LIN {X 0,Y 216.52,Z 296.519,A -85,B 0,C 180,E1 -21835.267,E2 -21835.267} C_VEL
LIN {X 0,Y 214.915,Z 310.205,A -85,B 0,C 180,E1 -21836.01,E2 -21836.01} C_VEL
LIN {X 0,Y 213.159,Z 322.237,A -85,B 0,C 180,E1 -21837.044,E2 -21837.044} C_VEL
LIN {X 0,Y 210.843,Z 333.547,A -85,B 0,C 180,E1 -21838.334,E2 -21838.334} C_VEL
LIN {X 0,Y 208.05,Z 345.191,A -85,B 0,C 180,E1 -21840.117,E2 -21840.117} C_VEL
LIN {X 0,Y 205.01,Z 355.654,A -85,B 0,C 180,E1 -21842.157,E2 -21842.157} C_VEL
LIN {X 0,Y 202.418,Z 364.207,A -85,B 0,C 180,E1 -21844.281,E2 -21844.281} C_VEL
LIN {X 0,Y 199.781,Z 372.178,A -85,B 0,C 180,E1 -21846.724,E2 -21846.724} C_VEL
LIN {X 0,Y 197.037,Z 379.781,A -85,B 0,C 180,E1 -21849.651,E2 -21849.651} C_VEL
LIN {X 0,Y 194.335,Z 386.855,A -85,B 0,C 180,E1 -21853.184,E2 -21853.184} C_VEL
LIN {X 0,Y 192.658,Z 391.564,A -85,B 0,C 180,E1 -21856.285,E2 -21856.285} C_VEL
LIN {X 0,Y 191.459,Z 395.168,A -85,B 0,C 180,E1 -21859.425,E2 -21859.425} C_VEL
LIN {X 0,Y 190.867,Z 397.03,A -85,B 0,C 180,E1 -21861.531,E2 -21861.531} C_VEL
LIN {X 0,Y 190.523,Z 398.428,A -85,B 0,C 180,E1 -21863.647,E2 -21863.647} C_VEL
LIN {X 0,Y 190.151,Z 400.035,A -85,B 0,C 180,E1 -21867.883,E2 -21867.883} C_VEL
LIN {X 0,Y 190.161,Z 400.264,A -85,B 0,C 180,E1 -21870.001,E2 -21870.001} C_VEL
LIN {X 0,Y 190.151,Z 400.068,A -85,B 0,C 180,E1 -21872.119,E2 -21872.119} C_VEL
LIN {X 0,Y 190.277,Z 399.478,A -85,B 0,C 180,E1 -21874.237,E2 -21874.237} C_VEL
LIN {X 0,Y 190.523,Z 398.504,A -85,B 0,C 180,E1 -21876.354,E2 -21876.354} C_VEL
LIN {X 0,Y 190.863,Z 397.139,A -85,B 0,C 180,E1 -21878.471,E2 -21878.471} C_VEL
LIN {X 0,Y 191.808,Z 394.255,A -85,B 0,C 180,E1 -21881.627,E2 -21881.627} C_VEL
LIN {X 0,Y 193.155,Z 390.346,A -85,B 0,C 180,E1 -21884.756,E2 -21884.756} C_VEL
LIN {X 0,Y 194.985,Z 385.304,A -85,B 0,C 180,E1 -21887.841,E2 -21887.841} C_VEL
LIN {X 0,Y 197.437,Z 378.955,A -85,B 0,C 180,E1 -21890.853,E2 -21890.853} C_VEL
LIN {X 0,Y 200.011,Z 371.649,A -85,B 0,C 180,E1 -21893.599,E2 -21893.599} C_VEL
LIN {X 0,Y 202.794,Z 362.923,A -85,B 0,C 180,E1 -21896.223,E2 -21896.223} C_VEL
LIN {X 0,Y 205.882,Z 353.047,A -85,B 0,C 180,E1 -21898.549,E2 -21898.549} C_VEL
LIN {X 0,Y 209.005,Z 341.929,A -85,B 0,C 180,E1 -21900.57,E2 -21900.57} C_VEL
LIN {X 0,Y 211.513,Z 331.031,A -85,B 0,C 180,E1 -21902.116,E2 -21902.116} C_VEL
LIN {X 0,Y 213.783,Z 318.986,A -85,B 0,C 180,E1 -21903.411,E2 -21903.411} C_VEL
LIN {X 0,Y 215.659,Z 305.842,A -85,B 0,C 180,E1 -21904.403,E2 -21904.403} C_VEL
LIN {X 0,Y 216.816,Z 292.984,A -85,B 0,C 180,E1 -21905.015,E2 -21905.015} C_VEL
LIN {X 0,Y 219.192,Z 241.525,A -85,B 0,C 180,E1 -21906.632,E2 -21906.632} C_VEL
LIN {X 0,Y 214.01,Z 228.643,A -85,B 0,C 180,E1 -21908.209,E2 -21908.209} C_VEL
LIN {X 0,Y 207.201,Z 214.231,A -85,B 0,C 180,E1 -21910.349,E2 -21910.349} C_VEL
LIN {X 0,Y 200.702,Z 202.668,A -85,B 0,C 180,E1 -21912.494,E2 -21912.494} C_VEL
LIN {X 0,Y 197.748,Z 198.045,A -85,B 0,C 180,E1 -21913.511,E2 -21913.511} C_VEL
LIN {X 0,Y 195.588,Z 194.613,A -85,B 0,C 180,E1 -21914.288,E2 -21914.288} C_VEL
LIN {X 0,Y 193.261,Z 191.834,A -85,B 0,C 180,E1 -21915.109,E2 -21915.109} C_VEL
LIN {X 0,Y 192.615,Z 190.071,A -85,B 0,C 180,E1 -21915.548,E2 -21915.548} C_VEL
LIN {X 0,Y 192.511,Z 189.538,A -85,B 0,C 180,E1 -21916.081,E2 -21916.081} C_VEL
LIN {X 0,Y 192.519,Z 189.499,A -85,B 0,C 180,E1 -21920.051,E2 -21920.051} C_VEL
LIN {X 0,Y 192.56,Z 189.439,A -85,B 0,C 180,E1 -21924.27,E2 -21924.27} C_VEL
LIN {X 0,Y 192.61,Z 189.447,A -85,B 0,C 180,E1 -21927.058,E2 -21927.058} C_VEL
LIN {X 0,Y 192.665,Z 189.47,A -85,B 0,C 180,E1 -21931.692,E2 -21931.692} C_VEL
LIN {X 0,Y 192.685,Z 189.474,A -85,B 0,C 180,E1 -21936.346,E2 -21936.346} C_VEL
LIN {X 0,Y 192.731,Z 189.477,A -85,B 0,C 180,E1 -21941.458,E2 -21941.458} C_VEL
LIN {X 0,Y 192.851,Z 189.461,A -85,B 0,C 180,E1 -21947.37,E2 -21947.37} C_VEL
LIN {X 0,Y 193.06,Z 189.411,A -85,B 0,C 180,E1 -21951.627,E2 -21951.627} C_VEL
LIN {X 0,Y 193.259,Z 189.386,A -85,B 0,C 180,E1 -21957.916,E2 -21957.916} C_VEL
LIN {X 0,Y 193.438,Z 189.382,A -85,B 0,C 180,E1 -21960,E2 -21960} C_VEL
LIN {X 0,Y 192.963,Z 189.423,A -85,B 0,C 180,E1 -21964.177,E2 -21964.177} C_VEL
LIN {X 0,Y 193.025,Z 189.441,A -85,B 0,C 180,E1 -21968.374,E2 -21968.374} C_VEL
LIN {X 0,Y 192.789,Z 189.451,A -85,B 0,C 180,E1 -21972.634,E2 -21972.634} C_VEL
LIN {X 0,Y 192.745,Z 189.456,A -85,B 0,C 180,E1 -21976.96,E2 -21976.96} C_VEL
LIN {X 0,Y 192.611,Z 189.492,A -85,B 0,C 180,E1 -21981.4,E2 -21981.4} C_VEL
LIN {X 0,Y 192.646,Z 189.469,A -85,B 0,C 180,E1 -21984.213,E2 -21984.213} C_VEL
LIN {X 0,Y 192.644,Z 189.473,A -85,B 0,C 180,E1 -21988.889,E2 -21988.889} C_VEL
LIN {X 0,Y 192.596,Z 189.478,A -85,B 0,C 180,E1 -21993.186,E2 -21993.186} C_VEL
LIN {X 0,Y 192.55,Z 189.454,A -85,B 0,C 180,E1 -21998.352,E2 -21998.352} C_VEL
LIN {X 0,Y 192.546,Z 189.606,A -85,B 0,C 180,E1 -22003.258,E2 -22003.258} C_VEL
LIN {X 0,Y 193.232,Z 191.826,A -85,B 0,C 180,E1 -22004.713,E2 -22004.713} C_VEL
LIN {X 0,Y 195.599,Z 195.89,A -85,B 0,C 180,E1 -22005.696,E2 -22005.696} C_VEL
LIN {X 0,Y 202.058,Z 206.618,A -85,B 0,C 180,E1 -22007.96,E2 -22007.96} C_VEL
LIN {X 0,Y 208.446,Z 218.785,A -85,B 0,C 180,E1 -22010.059,E2 -22010.059} C_VEL
LIN {X 0,Y 214.326,Z 231.789,A -85,B 0,C 180,E1 -22011.905,E2 -22011.905} C_VEL
LIN {X 0,Y 217.009,Z 238.438,A -85,B 0,C 180,E1 -22012.729,E2 -22012.729} C_VEL
LIN {X 0,Y 217.391,Z 241.526,A -85,B 0,C 180,E1 -22012.93,E2 -22012.93} C_VEL
LIN {X 0,Y 216.613,Z 246.06,A -85,B 0,C 180,E1 -22012.96,E2 -22012.96} C_VEL
LIN {X 0,Y 213.129,Z 256.558,A -85,B 0,C 180,E1 -22012.687,E2 -22012.687} C_VEL
LIN {X 0,Y 212.744,Z 259.307,A -85,B 0,C 180,E1 -22012.722,E2 -22012.722} C_VEL
LIN {X 0,Y 210.674,Z 300.138,A -85,B 0,C 180,E1 -22014.065,E2 -22014.065} C_VEL
LIN {X 0,Y 209.14,Z 313.363,A -85,B 0,C 180,E1 -22014.813,E2 -22014.813} C_VEL
LIN {X 0,Y 206.891,Z 326.323,A -85,B 0,C 180,E1 -22015.91,E2 -22015.91} C_VEL
LIN {X 0,Y 204.512,Z 337.393,A -85,B 0,C 180,E1 -22017.232,E2 -22017.232} C_VEL
LIN {X 0,Y 201.553,Z 348.935,A -85,B 0,C 180,E1 -22019.048,E2 -22019.048} C_VEL
LIN {X 0,Y 198.374,Z 359.328,A -85,B 0,C 180,E1 -22021.137,E2 -22021.137} C_VEL
LIN {X 0,Y 195.51,Z 367.823,A -85,B 0,C 180,E1 -22023.299,E2 -22023.299} C_VEL
LIN {X 0,Y 192.771,Z 375.975,A -85,B 0,C 180,E1 -22025.913,E2 -22025.913} C_VEL
LIN {X 0,Y 189.944,Z 383.312,A -85,B 0,C 180,E1 -22028.853,E2 -22028.853} C_VEL
LIN {X 0,Y 187.139,Z 390.37,A -85,B 0,C 180,E1 -22032.515,E2 -22032.515} C_VEL
LIN {X 0,Y 185.395,Z 395.063,A -85,B 0,C 180,E1 -22035.735,E2 -22035.735} C_VEL
LIN {X 0,Y 184.159,Z 398.646,A -85,B 0,C 180,E1 -22038.999,E2 -22038.999} C_VEL
LIN {X 0,Y 183.61,Z 400.493,A -85,B 0,C 180,E1 -22041.192,E2 -22041.192} C_VEL
LIN {X 0,Y 183.297,Z 401.878,A -85,B 0,C 180,E1 -22043.394,E2 -22043.394} C_VEL
LIN {X 0,Y 183.032,Z 403.227,A -85,B 0,C 180,E1 -22046.698,E2 -22046.698} C_VEL
LIN {X 0,Y 183.065,Z 403.678,A -85,B 0,C 180,E1 -22049.999,E2 -22049.999} C_VEL
LIN {X 0,Y 183.032,Z 403.215,A -85,B 0,C 180,E1 -22053.3,E2 -22053.3} C_VEL
LIN {X 0,Y 183.297,Z 401.849,A -85,B 0,C 180,E1 -22056.604,E2 -22056.604} C_VEL
LIN {X 0,Y 183.612,Z 400.45,A -85,B 0,C 180,E1 -22058.806,E2 -22058.806} C_VEL
LIN {X 0,Y 184.507,Z 397.518,A -85,B 0,C 180,E1 -22062.092,E2 -22062.092} C_VEL
LIN {X 0,Y 185.875,Z 393.55,A -85,B 0,C 180,E1 -22065.346,E2 -22065.346} C_VEL
LIN {X 0,Y 188.255,Z 387.448,A -85,B 0,C 180,E1 -22069.065,E2 -22069.065} C_VEL
LIN {X 0,Y 190.832,Z 380.783,A -85,B 0,C 180,E1 -22072.177,E2 -22072.177} C_VEL
LIN {X 0,Y 193.536,Z 373.421,A -85,B 0,C 180,E1 -22074.905,E2 -22074.905} C_VEL
LIN {X 0,Y 196.714,Z 364.027,A -85,B 0,C 180,E1 -22077.673,E2 -22077.673} C_VEL
LIN {X 0,Y 200.047,Z 353.54,A -85,B 0,C 180,E1 -22080.04,E2 -22080.04} C_VEL
LIN {X 0,Y 202.948,Z 343.16,A -85,B 0,C 180,E1 -22081.875,E2 -22081.875} C_VEL
LIN {X 0,Y 205.721,Z 331.768,A -85,B 0,C 180,E1 -22083.425,E2 -22083.425} C_VEL
LIN {X 0,Y 207.911,Z 320.025,A -85,B 0,C 180,E1 -22084.631,E2 -22084.631} C_VEL
LIN {X 0,Y 209.832,Z 306.994,A -85,B 0,C 180,E1 -22085.544,E2 -22085.544} C_VEL
LIN {X 0,Y 210.927,Z 294.034,A -85,B 0,C 180,E1 -22086.129,E2 -22086.129} C_VEL
LIN {X 0,Y 213.185,Z 246.397,A -85,B 0,C 180,E1 -22087.649,E2 -22087.649} C_VEL
LIN {X 0,Y 211.994,Z 242.409,A -85,B 0,C 180,E1 -22088.065,E2 -22088.065} C_VEL
LIN {X 0,Y 205.399,Z 226.595,A -85,B 0,C 180,E1 -22090.22,E2 -22090.22} C_VEL
LIN {X 0,Y 199.419,Z 214.433,A -85,B 0,C 180,E1 -22092.261,E2 -22092.261} C_VEL
LIN {X 0,Y 193.932,Z 204.867,A -85,B 0,C 180,E1 -22094.229,E2 -22094.229} C_VEL
LIN {X 0,Y 191.078,Z 200.191,A -85,B 0,C 180,E1 -22095.309,E2 -22095.309} C_VEL
LIN {X 0,Y 188.425,Z 196.048,A -85,B 0,C 180,E1 -22096.352,E2 -22096.352} C_VEL
LIN {X 0,Y 185.757,Z 191.777,A -85,B 0,C 180,E1 -22097.545,E2 -22097.545} C_VEL
LIN {X 0,Y 185.478,Z 190.463,A -85,B 0,C 180,E1 -22098.394,E2 -22098.394} C_VEL
LIN {X 0,Y 185.5,Z 190.321,A -85,B 0,C 180,E1 -22102.711,E2 -22102.711} C_VEL
LIN {X 0,Y 185.536,Z 190.375,A -85,B 0,C 180,E1 -22107.973,E2 -22107.973} C_VEL
LIN {X 0,Y 185.575,Z 190.352,A -85,B 0,C 180,E1 -22110.576,E2 -22110.576} C_VEL
LIN {X 0,Y 185.574,Z 190.35,A -85,B 0,C 180,E1 -22115.381,E2 -22115.381} C_VEL
LIN {X 0,Y 185.651,Z 190.339,A -85,B 0,C 180,E1 -22121.149,E2 -22121.149} C_VEL
LIN {X 0,Y 185.678,Z 190.354,A -85,B 0,C 180,E1 -22124.636,E2 -22124.636} C_VEL
LIN {X 0,Y 185.918,Z 190.303,A -85,B 0,C 180,E1 -22129.359,E2 -22129.359} C_VEL
LIN {X 0,Y 185.951,Z 190.307,A -85,B 0,C 180,E1 -22133.49,E2 -22133.49} C_VEL
LIN {X 0,Y 186.197,Z 190.285,A -85,B 0,C 180,E1 -22137.837,E2 -22137.837} C_VEL
LIN {X 0,Y 186.399,Z 190.259,A -85,B 0,C 180,E1 -22140,E2 -22140} C_VEL
LIN {X 0,Y 185.913,Z 190.313,A -85,B 0,C 180,E1 -22144.336,E2 -22144.336} C_VEL
LIN {X 0,Y 186.002,Z 190.289,A -85,B 0,C 180,E1 -22148.693,E2 -22148.693} C_VEL
LIN {X 0,Y 185.757,Z 190.344,A -85,B 0,C 180,E1 -22153.121,E2 -22153.121} C_VEL
LIN {X 0,Y 185.688,Z 190.356,A -85,B 0,C 180,E1 -22158.885,E2 -22158.885} C_VEL
LIN {X 0,Y 185.596,Z 190.366,A -85,B 0,C 180,E1 -22164.663,E2 -22164.663} C_VEL
LIN {X 0,Y 185.574,Z 190.361,A -85,B 0,C 180,E1 -22169.494,E2 -22169.494} C_VEL
LIN {X 0,Y 185.494,Z 190.318,A -85,B 0,C 180,E1 -22174.633,E2 -22174.633} C_VEL
LIN {X 0,Y 185.5,Z 190.331,A -85,B 0,C 180,E1 -22177.315,E2 -22177.315} C_VEL
LIN {X 0,Y 185.448,Z 190.501,A -85,B 0,C 180,E1 -22182.077,E2 -22182.077} C_VEL
LIN {X 0,Y 185.683,Z 191.483,A -85,B 0,C 180,E1 -22182.632,E2 -22182.632} C_VEL
LIN {X 0,Y 187.311,Z 194.335,A -85,B 0,C 180,E1 -22183.371,E2 -22183.371} C_VEL
LIN {X 0,Y 188.847,Z 195.941,A -85,B 0,C 180,E1 -22183.95,E2 -22183.95} C_VEL
LIN {X 0,Y 191.21,Z 199.43,A -85,B 0,C 180,E1 -22184.865,E2 -22184.865} C_VEL
LIN {X 0,Y 195.417,Z 205.792,A -85,B 0,C 180,E1 -22186.412,E2 -22186.412} C_VEL
LIN {X 0,Y 201.414,Z 216.342,A -85,B 0,C 180,E1 -22188.514,E2 -22188.514} C_VEL
LIN {X 0,Y 207.913,Z 229.985,A -85,B 0,C 180,E1 -22190.684,E2 -22190.684} C_VEL
LIN {X 0,Y 213.386,Z 243.368,A -85,B 0,C 180,E1 -22192.44,E2 -22192.44} C_VEL
LIN {X 0,Y 210.73,Z 296.676,A -85,B 0,C 180,E1 -22194.173,E2 -22194.173} C_VEL
LIN {X 0,Y 209.058,Z 310.386,A -85,B 0,C 180,E1 -22194.931,E2 -22194.931} C_VEL
LIN {X 0,Y 207.054,Z 323.393,A -85,B 0,C 180,E1 -22196.089,E2 -22196.089} C_VEL
LIN {X 0,Y 204.484,Z 335.201,A -85,B 0,C 180,E1 -22197.521,E2 -22197.521} C_VEL
LIN {X 0,Y 201.532,Z 346.551,A -85,B 0,C 180,E1 -22199.337,E2 -22199.337} C_VEL
LIN {X 0,Y 198.444,Z 356.78,A -85,B 0,C 180,E1 -22201.44,E2 -22201.44} C_VEL
LIN {X 0,Y 195.424,Z 366.126,A -85,B 0,C 180,E1 -22203.921,E2 -22203.921} C_VEL
LIN {X 0,Y 192.291,Z 374.888,A -85,B 0,C 180,E1 -22206.867,E2 -22206.867} C_VEL
LIN {X 0,Y 189.533,Z 382.075,A -85,B 0,C 180,E1 -22209.942,E2 -22209.942} C_VEL
LIN {X 0,Y 187.528,Z 386.921,A -85,B 0,C 180,E1 -22212.555,E2 -22212.555} C_VEL
LIN {X 0,Y 185.75,Z 391.631,A -85,B 0,C 180,E1 -22215.764,E2 -22215.764} C_VEL
LIN {X 0,Y 184.461,Z 395.234,A -85,B 0,C 180,E1 -22219.019,E2 -22219.019} C_VEL
LIN {X 0,Y 183.832,Z 397.096,A -85,B 0,C 180,E1 -22221.205,E2 -22221.205} C_VEL
LIN {X 0,Y 183.448,Z 398.494,A -85,B 0,C 180,E1 -22223.401,E2 -22223.401} C_VEL
LIN {X 0,Y 183.097,Z 399.767,A -85,B 0,C 180,E1 -22226.367,E2 -22226.367} C_VEL
LIN {X 0,Y 183.072,Z 400.329,A -85,B 0,C 180,E1 -22230.001,E2 -22230.001} C_VEL
LIN {X 0,Y 183.154,Z 399.723,A -85,B 0,C 180,E1 -22233.906,E2 -22233.906} C_VEL
LIN {X 0,Y 183.448,Z 398.569,A -85,B 0,C 180,E1 -22236.6,E2 -22236.6} C_VEL
LIN {X 0,Y 183.829,Z 397.204,A -85,B 0,C 180,E1 -22238.797,E2 -22238.797} C_VEL
LIN {X 0,Y 184.841,Z 394.319,A -85,B 0,C 180,E1 -22242.071,E2 -22242.071} C_VEL
LIN {X 0,Y 186.272,Z 390.41,A -85,B 0,C 180,E1 -22245.315,E2 -22245.315} C_VEL
LIN {X 0,Y 188.219,Z 385.368,A -85,B 0,C 180,E1 -22248.505,E2 -22248.505} C_VEL
LIN {X 0,Y 190.8,Z 379.018,A -85,B 0,C 180,E1 -22251.614,E2 -22251.614} C_VEL
LIN {X 0,Y 193.325,Z 372.255,A -85,B 0,C 180,E1 -22254.258,E2 -22254.258} C_VEL
LIN {X 0,Y 196.444,Z 362.985,A -85,B 0,C 180,E1 -22257.139,E2 -22257.139} C_VEL
LIN {X 0,Y 199.684,Z 353.109,A -85,B 0,C 180,E1 -22259.521,E2 -22259.521} C_VEL
LIN {X 0,Y 202.918,Z 341.989,A -85,B 0,C 180,E1 -22261.591,E2 -22261.591} C_VEL
LIN {X 0,Y 205.529,Z 331.09,A -85,B 0,C 180,E1 -22263.169,E2 -22263.169} C_VEL
LIN {X 0,Y 207.889,Z 319.043,A -85,B 0,C 180,E1 -22264.49,E2 -22264.49} C_VEL
LIN {X 0,Y 209.796,Z 306.311,A -85,B 0,C 180,E1 -22265.474,E2 -22265.474} C_VEL
LIN {X 0,Y 211.048,Z 293.249,A -85,B 0,C 180,E1 -22266.109,E2 -22266.109} C_VEL
LIN {X 0,Y 213.46,Z 243.344,A -85,B 0,C 180,E1 -22267.711,E2 -22267.711} C_VEL
LIN {X 0,Y 208.208,Z 230.53,A -85,B 0,C 180,E1 -22269.397,E2 -22269.397} C_VEL
LIN {X 0,Y 202.113,Z 217.696,A -85,B 0,C 180,E1 -22271.426,E2 -22271.426} C_VEL
LIN {X 0,Y 196.616,Z 207.676,A -85,B 0,C 180,E1 -22273.349,E2 -22273.349} C_VEL
LIN {X 0,Y 193.586,Z 202.92,A -85,B 0,C 180,E1 -22274.445,E2 -22274.445} C_VEL
LIN {X 0,Y 191.026,Z 199.227,A -85,B 0,C 180,E1 -22275.397,E2 -22275.397} C_VEL
LIN {X 0,Y 188.755,Z 195.702,A -85,B 0,C 180,E1 -22276.292,E2 -22276.292} C_VEL
LIN {X 0,Y 186.317,Z 192.945,A -85,B 0,C 180,E1 -22277.236,E2 -22277.236} C_VEL
LIN {X 0,Y 185.532,Z 190.905,A -85,B 0,C 180,E1 -22277.792,E2 -22277.792} C_VEL
LIN {X 0,Y 185.452,Z 190.446,A -85,B 0,C 180,E1 -22278.233,E2 -22278.233} C_VEL
LIN {X 0,Y 185.506,Z 190.333,A -85,B 0,C 180,E1 -22282.712,E2 -22282.712} C_VEL
LIN {X 0,Y 185.546,Z 190.342,A -85,B 0,C 180,E1 -22287.975,E2 -22287.975} C_VEL
LIN {X 0,Y 185.582,Z 190.361,A -85,B 0,C 180,E1 -22290.576,E2 -22290.576} C_VEL
LIN {X 0,Y 185.58,Z 190.369,A -85,B 0,C 180,E1 -22295.381,E2 -22295.381} C_VEL
LIN {X 0,Y 185.674,Z 190.357,A -85,B 0,C 180,E1 -22301.134,E2 -22301.134} C_VEL
LIN {X 0,Y 185.762,Z 190.342,A -85,B 0,C 180,E1 -22306.879,E2 -22306.879} C_VEL
LIN {X 0,Y 186.008,Z 190.288,A -85,B 0,C 180,E1 -22311.307,E2 -22311.307} C_VEL
LIN {X 0,Y 186.204,Z 190.264,A -85,B 0,C 180,E1 -22317.837,E2 -22317.837} C_VEL
LIN {X 0,Y 186.402,Z 190.258,A -85,B 0,C 180,E1 -22320,E2 -22320} C_VEL
LIN {X 0,Y 185.909,Z 190.301,A -85,B 0,C 180,E1 -22324.336,E2 -22324.336} C_VEL
LIN {X 0,Y 185.974,Z 190.317,A -85,B 0,C 180,E1 -22328.694,E2 -22328.694} C_VEL
LIN {X 0,Y 185.717,Z 190.337,A -85,B 0,C 180,E1 -22333.124,E2 -22333.124} C_VEL
LIN {X 0,Y 185.683,Z 190.333,A -85,B 0,C 180,E1 -22337.626,E2 -22337.626} C_VEL
LIN {X 0,Y 185.574,Z 190.358,A -85,B 0,C 180,E1 -22342.254,E2 -22342.254} C_VEL
LIN {X 0,Y 185.558,Z 190.372,A -85,B 0,C 180,E1 -22347.033,E2 -22347.033} C_VEL
LIN {X 0,Y 185.577,Z 190.352,A -85,B 0,C 180,E1 -22349.493,E2 -22349.493} C_VEL
LIN {X 0,Y 185.498,Z 190.333,A -85,B 0,C 180,E1 -22354.632,E2 -22354.632} C_VEL
LIN {X 0,Y 185.504,Z 190.321,A -85,B 0,C 180,E1 -22357.314,E2 -22357.314} C_VEL
LIN {X 0,Y 185.476,Z 190.553,A -85,B 0,C 180,E1 -22361.606,E2 -22361.606} C_VEL
LIN {X 0,Y 185.867,Z 192.023,A -85,B 0,C 180,E1 -22362.424,E2 -22362.424} C_VEL
LIN {X 0,Y 189.734,Z 197.961,A -85,B 0,C 180,E1 -22364.054,E2 -22364.054} C_VEL
LIN {X 0,Y 195.512,Z 207.366,A -85,B 0,C 180,E1 -22366.245,E2 -22366.245} C_VEL
LIN {X 0,Y 202.294,Z 219.885,A -85,B 0,C 180,E1 -22368.637,E2 -22368.637} C_VEL
LIN {X 0,Y 208.335,Z 233.114,A -85,B 0,C 180,E1 -22370.661,E2 -22370.661} C_VEL
LIN {X 0,Y 213.143,Z 245.402,A -85,B 0,C 180,E1 -22372.226,E2 -22372.226} C_VEL
LIN {X 0,Y 213.37,Z 248.029,A -85,B 0,C 180,E1 -22372.382,E2 -22372.382} C_VEL
LIN {X 0,Y 212.744,Z 259.307,A -85,B 0,C 180,E1 -22372.722,E2 -22372.722} C_VEL
LIN {X 0,Y 211.928,Z 265.149,A -85,B 0,C 180,E1 -22372.798,E2 -22372.798} C_VEL
LIN {X 0,Y 206.47,Z 284.171,A -85,B 0,C 180,E1 -22372.463,E2 -22372.463} C_VEL
LIN {X 0,Y 205.612,Z 290.015,A -85,B 0,C 180,E1 -22372.531,E2 -22372.531} C_VEL
LIN {X 0,Y 204.494,Z 304.483,A -85,B 0,C 180,E1 -22373.099,E2 -22373.099} C_VEL
LIN {X 0,Y 202.62,Z 318.008,A -85,B 0,C 180,E1 -22374.021,E2 -22374.021} C_VEL
LIN {X 0,Y 200.206,Z 330.248,A -85,B 0,C 180,E1 -22375.219,E2 -22375.219} C_VEL
LIN {X 0,Y 197.428,Z 342.014,A -85,B 0,C 180,E1 -22376.817,E2 -22376.817} C_VEL
LIN {X 0,Y 193.965,Z 353.761,A -85,B 0,C 180,E1 -22378.914,E2 -22378.914} C_VEL
LIN {X 0,Y 190.484,Z 364.189,A -85,B 0,C 180,E1 -22381.338,E2 -22381.338} C_VEL
LIN {X 0,Y 187.472,Z 372.497,A -85,B 0,C 180,E1 -22383.812,E2 -22383.812} C_VEL
LIN {X 0,Y 184.282,Z 380.866,A -85,B 0,C 180,E1 -22386.989,E2 -22386.989} C_VEL
LIN {X 0,Y 181.564,Z 387.503,A -85,B 0,C 180,E1 -22390.202,E2 -22390.202} C_VEL
LIN {X 0,Y 179.008,Z 393.571,A -85,B 0,C 180,E1 -22394.048,E2 -22394.048} C_VEL
LIN {X 0,Y 177.542,Z 397.515,A -85,B 0,C 180,E1 -22397.424,E2 -22397.424} C_VEL
LIN {X 0,Y 176.585,Z 400.429,A -85,B 0,C 180,E1 -22400.839,E2 -22400.839} C_VEL
LIN {X 0,Y 176.235,Z 401.814,A -85,B 0,C 180,E1 -22403.128,E2 -22403.128} C_VEL
LIN {X 0,Y 175.911,Z 403.295,A -85,B 0,C 180,E1 -22407.194,E2 -22407.194} C_VEL
LIN {X 0,Y 175.977,Z 403.614,A -85,B 0,C 180,E1 -22409.999,E2 -22409.999} C_VEL
LIN {X 0,Y 175.911,Z 403.282,A -85,B 0,C 180,E1 -22412.804,E2 -22412.804} C_VEL
LIN {X 0,Y 176.234,Z 401.783,A -85,B 0,C 180,E1 -22416.87,E2 -22416.87} C_VEL
LIN {X 0,Y 176.587,Z 400.385,A -85,B 0,C 180,E1 -22419.159,E2 -22419.159} C_VEL
LIN {X 0,Y 177.546,Z 397.452,A -85,B 0,C 180,E1 -22422.573,E2 -22422.573} C_VEL
LIN {X 0,Y 179.004,Z 393.484,A -85,B 0,C 180,E1 -22425.951,E2 -22425.951} C_VEL
LIN {X 0,Y 181.553,Z 387.382,A -85,B 0,C 180,E1 -22429.797,E2 -22429.797} C_VEL
LIN {X 0,Y 184.274,Z 380.717,A -85,B 0,C 180,E1 -22433.01,E2 -22433.01} C_VEL
LIN {X 0,Y 187.466,Z 372.313,A -85,B 0,C 180,E1 -22436.187,E2 -22436.187} C_VEL
LIN {X 0,Y 190.44,Z 363.959,A -85,B 0,C 180,E1 -22438.667,E2 -22438.667} C_VEL
LIN {X 0,Y 193.904,Z 353.471,A -85,B 0,C 180,E1 -22441.095,E2 -22441.095} C_VEL
LIN {X 0,Y 196.967,Z 343.091,A -85,B 0,C 180,E1 -22442.964,E2 -22442.964} C_VEL
LIN {X 0,Y 199.838,Z 331.697,A -85,B 0,C 180,E1 -22444.546,E2 -22444.546} C_VEL
LIN {X 0,Y 202.119,Z 319.952,A -85,B 0,C 180,E1 -22445.773,E2 -22445.773} C_VEL
LIN {X 0,Y 204.132,Z 306.763,A -85,B 0,C 180,E1 -22446.708,E2 -22446.708} C_VEL
LIN {X 0,Y 205.22,Z 294.43,A -85,B 0,C 180,E1 -22447.276,E2 -22447.276} C_VEL
LIN {X 0,Y 207.579,Z 247.803,A -85,B 0,C 180,E1 -22448.788,E2 -22448.788} C_VEL
LIN {X 0,Y 201.592,Z 232.687,A -85,B 0,C 180,E1 -22450.857,E2 -22450.857} C_VEL
LIN {X 0,Y 196.18,Z 221.24,A -85,B 0,C 180,E1 -22452.791,E2 -22452.791} C_VEL
LIN {X 0,Y 190.505,Z 210.736,A -85,B 0,C 180,E1 -22454.931,E2 -22454.931} C_VEL
LIN {X 0,Y 185.027,Z 201.72,A -85,B 0,C 180,E1 -22457.145,E2 -22457.145} C_VEL
LIN {X 0,Y 181.266,Z 196.109,A -85,B 0,C 180,E1 -22458.767,E2 -22458.767} C_VEL
LIN {X 0,Y 179.331,Z 193.911,A -85,B 0,C 180,E1 -22459.608,E2 -22459.608} C_VEL
LIN {X 0,Y 178.511,Z 191.858,A -85,B 0,C 180,E1 -22460.226,E2 -22460.226} C_VEL
LIN {X 0,Y 178.389,Z 191.283,A -85,B 0,C 180,E1 -22460.924,E2 -22460.924} C_VEL
LIN {X 0,Y 178.478,Z 191.213,A -85,B 0,C 180,E1 -22465.78,E2 -22465.78} C_VEL
LIN {X 0,Y 178.516,Z 191.232,A -85,B 0,C 180,E1 -22470.006,E2 -22470.006} C_VEL
LIN {X 0,Y 178.514,Z 191.232,A -85,B 0,C 180,E1 -22474.885,E2 -22474.885} C_VEL
LIN {X 0,Y 178.603,Z 191.219,A -85,B 0,C 180,E1 -22480.797,E2 -22480.797} C_VEL
LIN {X 0,Y 178.646,Z 191.223,A -85,B 0,C 180,E1 -22486.347,E2 -22486.347} C_VEL
LIN {X 0,Y 178.952,Z 191.188,A -85,B 0,C 180,E1 -22490.962,E2 -22490.962} C_VEL
LIN {X 0,Y 179.143,Z 191.162,A -85,B 0,C 180,E1 -22497.752,E2 -22497.752} C_VEL
LIN {X 0,Y 179.362,Z 191.135,A -85,B 0,C 180,E1 -22500,E2 -22500} C_VEL
LIN {X 0,Y 178.861,Z 191.193,A -85,B 0,C 180,E1 -22504.507,E2 -22504.507} C_VEL
LIN {X 0,Y 178.931,Z 191.168,A -85,B 0,C 180,E1 -22509.039,E2 -22509.039} C_VEL
LIN {X 0,Y 178.675,Z 191.219,A -85,B 0,C 180,E1 -22513.651,E2 -22513.651} C_VEL
LIN {X 0,Y 178.633,Z 191.234,A -85,B 0,C 180,E1 -22519.231,E2 -22519.231} C_VEL
LIN {X 0,Y 178.529,Z 191.248,A -85,B 0,C 180,E1 -22525.125,E2 -22525.125} C_VEL
LIN {X 0,Y 178.496,Z 191.25,A -85,B 0,C 180,E1 -22530.788,E2 -22530.788} C_VEL
LIN {X 0,Y 178.48,Z 191.192,A -85,B 0,C 180,E1 -22534.221,E2 -22534.221} C_VEL
LIN {X 0,Y 178.433,Z 191.413,A -85,B 0,C 180,E1 -22539.612,E2 -22539.612} C_VEL
LIN {X 0,Y 178.678,Z 192.427,A -85,B 0,C 180,E1 -22540.189,E2 -22540.189} C_VEL
LIN {X 0,Y 180.292,Z 195.247,A -85,B 0,C 180,E1 -22541.002,E2 -22541.002} C_VEL
LIN {X 0,Y 181.843,Z 196.704,A -85,B 0,C 180,E1 -22541.648,E2 -22541.648} C_VEL
LIN {X 0,Y 184.137,Z 200.235,A -85,B 0,C 180,E1 -22542.646,E2 -22542.646} C_VEL
LIN {X 0,Y 185.481,Z 201.977,A -85,B 0,C 180,E1 -22543.193,E2 -22543.193} C_VEL
LIN {X 0,Y 190.843,Z 209.804,A -85,B 0,C 180,E1 -22545.295,E2 -22545.295} C_VEL
LIN {X 0,Y 197.056,Z 220.991,A -85,B 0,C 180,E1 -22547.605,E2 -22547.605} C_VEL
LIN {X 0,Y 203.025,Z 233.783,A -85,B 0,C 180,E1 -22549.714,E2 -22549.714} C_VEL
LIN {X 0,Y 207.716,Z 245.315,A -85,B 0,C 180,E1 -22551.308,E2 -22551.308} C_VEL
LIN {X 0,Y 204.988,Z 296.952,A -85,B 0,C 180,E1 -22553.019,E2 -22553.019} C_VEL
LIN {X 0,Y 203.279,Z 310.571,A -85,B 0,C 180,E1 -22553.791,E2 -22553.791} C_VEL
LIN {X 0,Y 201.192,Z 323.464,A -85,B 0,C 180,E1 -22554.959,E2 -22554.959} C_VEL
LIN {X 0,Y 198.525,Z 335.271,A -85,B 0,C 180,E1 -22556.419,E2 -22556.419} C_VEL
LIN {X 0,Y 195.457,Z 346.62,A -85,B 0,C 180,E1 -22558.275,E2 -22558.275} C_VEL
LIN {X 0,Y 192.222,Z 356.848,A -85,B 0,C 180,E1 -22560.425,E2 -22560.425} C_VEL
LIN {X 0,Y 189.115,Z 366.03,A -85,B 0,C 180,E1 -22562.921,E2 -22562.921} C_VEL
LIN {X 0,Y 185.753,Z 374.956,A -85,B 0,C 180,E1 -22566.002,E2 -22566.002} C_VEL
LIN {X 0,Y 182.873,Z 382.142,A -85,B 0,C 180,E1 -22569.178,E2 -22569.178} C_VEL
LIN {X 0,Y 180.743,Z 386.988,A -85,B 0,C 180,E1 -22571.878,E2 -22571.878} C_VEL
LIN {X 0,Y 178.866,Z 391.697,A -85,B 0,C 180,E1 -22575.204,E2 -22575.204} C_VEL
LIN {X 0,Y 177.486,Z 395.3,A -85,B 0,C 180,E1 -22578.582,E2 -22578.582} C_VEL
LIN {X 0,Y 176.818,Z 397.161,A -85,B 0,C 180,E1 -22580.853,E2 -22580.853} C_VEL
LIN {X 0,Y 176.399,Z 398.559,A -85,B 0,C 180,E1 -22583.136,E2 -22583.136} C_VEL
LIN {X 0,Y 175.996,Z 399.951,A -85,B 0,C 180,E1 -22586.682,E2 -22586.682} C_VEL
LIN {X 0,Y 175.985,Z 400.394,A -85,B 0,C 180,E1 -22590.001,E2 -22590.001} C_VEL
LIN {X 0,Y 176.003,Z 399.975,A -85,B 0,C 180,E1 -22593.356,E2 -22593.356} C_VEL
LIN {X 0,Y 176.398,Z 398.633,A -85,B 0,C 180,E1 -22596.866,E2 -22596.866} C_VEL
LIN {X 0,Y 176.816,Z 397.268,A -85,B 0,C 180,E1 -22599.149,E2 -22599.149} C_VEL
LIN {X 0,Y 177.897,Z 394.384,A -85,B 0,C 180,E1 -22602.55,E2 -22602.55} C_VEL
LIN {X 0,Y 179.416,Z 390.474,A -85,B 0,C 180,E1 -22605.915,E2 -22605.915} C_VEL
LIN {X 0,Y 181.487,Z 385.431,A -85,B 0,C 180,E1 -22609.218,E2 -22609.218} C_VEL
LIN {X 0,Y 184.198,Z 379.081,A -85,B 0,C 180,E1 -22612.43,E2 -22612.43} C_VEL
LIN {X 0,Y 187.331,Z 371.069,A -85,B 0,C 180,E1 -22615.588,E2 -22615.588} C_VEL
LIN {X 0,Y 190.773,Z 361.266,A -85,B 0,C 180,E1 -22618.615,E2 -22618.615} C_VEL
LIN {X 0,Y 194.27,Z 350.894,A -85,B 0,C 180,E1 -22621.032,E2 -22621.032} C_VEL
LIN {X 0,Y 197.677,Z 339.2,A -85,B 0,C 180,E1 -22623.136,E2 -22623.136} C_VEL
LIN {X 0,Y 200.469,Z 327.53,A -85,B 0,C 180,E1 -22624.729,E2 -22624.729} C_VEL
LIN {X 0,Y 202.732,Z 315.389,A -85,B 0,C 180,E1 -22625.956,E2 -22625.956} C_VEL
LIN {X 0,Y 204.591,Z 301.911,A -85,B 0,C 180,E1 -22626.892,E2 -22626.892} C_VEL
LIN {X 0,Y 205.592,Z 287.978,A -85,B 0,C 180,E1 -22627.477,E2 -22627.477} C_VEL
LIN {X 0,Y 207.789,Z 245.398,A -85,B 0,C 180,E1 -22628.842,E2 -22628.842} C_VEL
LIN {X 0,Y 202.79,Z 233.044,A -85,B 0,C 180,E1 -22630.552,E2 -22630.552} C_VEL
LIN {X 0,Y 196.691,Z 220.188,A -85,B 0,C 180,E1 -22632.716,E2 -22632.716} C_VEL
LIN {X 0,Y 190.387,Z 208.988,A -85,B 0,C 180,E1 -22635.079,E2 -22635.079} C_VEL
LIN {X 0,Y 186.886,Z 204.054,A -85,B 0,C 180,E1 -22636.437,E2 -22636.437} C_VEL
LIN {X 0,Y 184.579,Z 200.658,A -85,B 0,C 180,E1 -22637.387,E2 -22637.387} C_VEL
LIN {X 0,Y 182.217,Z 197.445,A -85,B 0,C 180,E1 -22638.388,E2 -22638.388} C_VEL
LIN {X 0,Y 181.595,Z 196.371,A -85,B 0,C 180,E1 -22638.673,E2 -22638.673} C_VEL
LIN {X 0,Y 179.388,Z 194.013,A -85,B 0,C 180,E1 -22639.626,E2 -22639.626} C_VEL
LIN {X 0,Y 178.502,Z 191.828,A -85,B 0,C 180,E1 -22640.269,E2 -22640.269} C_VEL
LIN {X 0,Y 178.396,Z 191.305,A -85,B 0,C 180,E1 -22640.925,E2 -22640.925} C_VEL
LIN {X 0,Y 178.485,Z 191.191,A -85,B 0,C 180,E1 -22645.781,E2 -22645.781} C_VEL
LIN {X 0,Y 178.523,Z 191.247,A -85,B 0,C 180,E1 -22650.006,E2 -22650.006} C_VEL
LIN {X 0,Y 178.52,Z 191.249,A -85,B 0,C 180,E1 -22654.886,E2 -22654.886} C_VEL
LIN {X 0,Y 178.622,Z 191.235,A -85,B 0,C 180,E1 -22660.785,E2 -22660.785} C_VEL
LIN {X 0,Y 178.679,Z 191.217,A -85,B 0,C 180,E1 -22666.349,E2 -22666.349} C_VEL
LIN {X 0,Y 178.937,Z 191.168,A -85,B 0,C 180,E1 -22670.961,E2 -22670.961} C_VEL
LIN {X 0,Y 179.149,Z 191.142,A -85,B 0,C 180,E1 -22677.752,E2 -22677.752} C_VEL
LIN {X 0,Y 179.365,Z 191.134,A -85,B 0,C 180,E1 -22680,E2 -22680} C_VEL
LIN {X 0,Y 178.857,Z 191.179,A -85,B 0,C 180,E1 -22684.507,E2 -22684.507} C_VEL
LIN {X 0,Y 178.904,Z 191.193,A -85,B 0,C 180,E1 -22689.041,E2 -22689.041} C_VEL
LIN {X 0,Y 178.646,Z 191.224,A -85,B 0,C 180,E1 -22693.653,E2 -22693.653} C_VEL
LIN {X 0,Y 178.609,Z 191.219,A -85,B 0,C 180,E1 -22699.203,E2 -22699.203} C_VEL
LIN {X 0,Y 178.519,Z 191.233,A -85,B 0,C 180,E1 -22705.114,E2 -22705.114} C_VEL
LIN {X 0,Y 178.521,Z 191.232,A -85,B 0,C 180,E1 -22709.993,E2 -22709.993} C_VEL
LIN {X 0,Y 178.483,Z 191.211,A -85,B 0,C 180,E1 -22714.219,E2 -22714.219} C_VEL
LIN {X 0,Y 178.408,Z 191.393,A -85,B 0,C 180,E1 -22719.253,E2 -22719.253} C_VEL
LIN {X 0,Y 178.634,Z 192.298,A -85,B 0,C 180,E1 -22719.833,E2 -22719.833} C_VEL
LIN {X 0,Y 180.216,Z 195.158,A -85,B 0,C 180,E1 -22720.669,E2 -22720.669} C_VEL
LIN {X 0,Y 181.959,Z 196.997,A -85,B 0,C 180,E1 -22721.41,E2 -22721.41} C_VEL
LIN {X 0,Y 186.389,Z 203.956,A -85,B 0,C 180,E1 -22723.313,E2 -22723.313} C_VEL
LIN {X 0,Y 191.122,Z 211.682,A -85,B 0,C 180,E1 -22725.198,E2 -22725.198} C_VEL
LIN {X 0,Y 197.898,Z 224.526,A -85,B 0,C 180,E1 -22727.731,E2 -22727.731} C_VEL
LIN {X 0,Y 203.551,Z 237.203,A -85,B 0,C 180,E1 -22729.736,E2 -22729.736} C_VEL
LIN {X 0,Y 207.701,Z 247.904,A -85,B 0,C 180,E1 -22731.164,E2 -22731.164} C_VEL
LIN {X 0,Y 205.612,Z 290.015,A -85,B 0,C 180,E1 -22732.531,E2 -22732.531} C_VEL
LIN {X 0,Y 204.661,Z 295.846,A -85,B 0,C 180,E1 -22732.594,E2 -22732.594} C_VEL
LIN {X 0,Y 201.448,Z 305.24,A -85,B 0,C 180,E1 -22732.511,E2 -22732.511} C_VEL
LIN {X 0,Y 197.96,Z 314.534,A -85,B 0,C 180,E1 -22732.632,E2 -22732.632} C_VEL
LIN {X 0,Y 196.54,Z 320.102,A -85,B 0,C 180,E1 -22732.99,E2 -22732.99} C_VEL
LIN {X 0,Y 193.987,Z 332.079,A -85,B 0,C 180,E1 -22734.254,E2 -22734.254} C_VEL
LIN {X 0,Y 191.09,Z 343.38,A -85,B 0,C 180,E1 -22735.884,E2 -22735.884} C_VEL
LIN {X 0,Y 187.918,Z 353.7,A -85,B 0,C 180,E1 -22737.795,E2 -22737.795} C_VEL
LIN {X 0,Y 184.261,Z 364.126,A -85,B 0,C 180,E1 -22740.274,E2 -22740.274} C_VEL
LIN {X 0,Y 181.049,Z 372.566,A -85,B 0,C 180,E1 -22742.864,E2 -22742.864} C_VEL
LIN {X 0,Y 177.769,Z 380.803,A -85,B 0,C 180,E1 -22746.094,E2 -22746.094} C_VEL
LIN {X 0,Y 174.892,Z 387.44,A -85,B 0,C 180,E1 -22749.413,E2 -22749.413} C_VEL
LIN {X 0,Y 172.159,Z 393.507,A -85,B 0,C 180,E1 -22753.395,E2 -22753.395} C_VEL
LIN {X 0,Y 170.606,Z 397.451,A -85,B 0,C 180,E1 -22756.904,E2 -22756.904} C_VEL
LIN {X 0,Y 169.555,Z 400.364,A -85,B 0,C 180,E1 -22760.456,E2 -22760.456} C_VEL
LIN {X 0,Y 169.167,Z 401.749,A -85,B 0,C 180,E1 -22762.84,E2 -22762.84} C_VEL
LIN {X 0,Y 168.937,Z 402.737,A -85,B 0,C 180,E1 -22765.226,E2 -22765.226} C_VEL
LIN {X 0,Y 168.819,Z 403.339,A -85,B 0,C 180,E1 -22767.613,E2 -22767.613} C_VEL
LIN {X 0,Y 168.875,Z 403.549,A -85,B 0,C 180,E1 -22769.999,E2 -22769.999} C_VEL
LIN {X 0,Y 168.819,Z 403.325,A -85,B 0,C 180,E1 -22772.385,E2 -22772.385} C_VEL
LIN {X 0,Y 168.936,Z 402.715,A -85,B 0,C 180,E1 -22774.772,E2 -22774.772} C_VEL
LIN {X 0,Y 169.167,Z 401.718,A -85,B 0,C 180,E1 -22777.158,E2 -22777.158} C_VEL
LIN {X 0,Y 169.557,Z 400.319,A -85,B 0,C 180,E1 -22779.542,E2 -22779.542} C_VEL
LIN {X 0,Y 170.608,Z 397.386,A -85,B 0,C 180,E1 -22783.094,E2 -22783.094} C_VEL
LIN {X 0,Y 172.155,Z 393.417,A -85,B 0,C 180,E1 -22786.603,E2 -22786.603} C_VEL
LIN {X 0,Y 174.882,Z 387.315,A -85,B 0,C 180,E1 -22790.586,E2 -22790.586} C_VEL
LIN {X 0,Y 177.762,Z 380.65,A -85,B 0,C 180,E1 -22793.905,E2 -22793.905} C_VEL
LIN {X 0,Y 180.978,Z 372.527,A -85,B 0,C 180,E1 -22797.084,E2 -22797.084} C_VEL
LIN {X 0,Y 184.236,Z 363.891,A -85,B 0,C 180,E1 -22799.728,E2 -22799.728} C_VEL
LIN {X 0,Y 187.857,Z 353.403,A -85,B 0,C 180,E1 -22802.214,E2 -22802.214} C_VEL
LIN {X 0,Y 191.052,Z 343.021,A -85,B 0,C 180,E1 -22804.122,E2 -22804.122} C_VEL
LIN {X 0,Y 194.041,Z 331.627,A -85,B 0,C 180,E1 -22805.733,E2 -22805.733} C_VEL
LIN {X 0,Y 196.408,Z 319.879,A -85,B 0,C 180,E1 -22806.982,E2 -22806.982} C_VEL
LIN {X 0,Y 198.489,Z 306.631,A -85,B 0,C 180,E1 -22807.938,E2 -22807.938} C_VEL
LIN {X 0,Y 199.666,Z 293.546,A -85,B 0,C 180,E1 -22808.542,E2 -22808.542} C_VEL
LIN {X 0,Y 202.044,Z 249.853,A -85,B 0,C 180,E1 -22809.964,E2 -22809.964} C_VEL
LIN {X 0,Y 196.234,Z 235.281,A -85,B 0,C 180,E1 -22812.095,E2 -22812.095} C_VEL
LIN {X 0,Y 190.857,Z 223.703,A -85,B 0,C 180,E1 -22814.157,E2 -22814.157} C_VEL
LIN {X 0,Y 184.016,Z 211.302,A -85,B 0,C 180,E1 -22816.946,E2 -22816.946} C_VEL
LIN {X 0,Y 178.135,Z 202.025,A -85,B 0,C 180,E1 -22819.565,E2 -22819.565} C_VEL
LIN {X 0,Y 175.759,Z 199.136,A -85,B 0,C 180,E1 -22820.662,E2 -22820.662} C_VEL
LIN {X 0,Y 174.833,Z 197.414,A -85,B 0,C 180,E1 -22821.142,E2 -22821.142} C_VEL
LIN {X 0,Y 172.619,Z 195.298,A -85,B 0,C 180,E1 -22822.201,E2 -22822.201} C_VEL
LIN {X 0,Y 171.498,Z 192.816,A -85,B 0,C 180,E1 -22822.994,E2 -22822.994} C_VEL
LIN {X 0,Y 171.393,Z 192.132,A -85,B 0,C 180,E1 -22823.7,E2 -22823.7} C_VEL
LIN {X 0,Y 171.434,Z 192.117,A -85,B 0,C 180,E1 -22829.414,E2 -22829.414} C_VEL
LIN {X 0,Y 171.452,Z 192.116,A -85,B 0,C 180,E1 -22834.391,E2 -22834.391} C_VEL
LIN {X 0,Y 171.559,Z 192.096,A -85,B 0,C 180,E1 -22840.869,E2 -22840.869} C_VEL
LIN {X 0,Y 171.564,Z 192.112,A -85,B 0,C 180,E1 -22845.772,E2 -22845.772} C_VEL
LIN {X 0,Y 171.881,Z 192.062,A -85,B 0,C 180,E1 -22850.587,E2 -22850.587} C_VEL
LIN {X 0,Y 171.808,Z 192.056,A -85,B 0,C 180,E1 -22855.307,E2 -22855.307} C_VEL
LIN {X 0,Y 172.325,Z 192.01,A -85,B 0,C 180,E1 -22860,E2 -22860} C_VEL
LIN {X 0,Y 171.811,Z 192.073,A -85,B 0,C 180,E1 -22864.693,E2 -22864.693} C_VEL
LIN {X 0,Y 171.867,Z 192.048,A -85,B 0,C 180,E1 -22869.414,E2 -22869.414} C_VEL
LIN {X 0,Y 171.59,Z 192.093,A -85,B 0,C 180,E1 -22874.226,E2 -22874.226} C_VEL
LIN {X 0,Y 171.552,Z 192.113,A -85,B 0,C 180,E1 -22879.575,E2 -22879.575} C_VEL
LIN {X 0,Y 171.464,Z 192.123,A -85,B 0,C 180,E1 -22885.617,E2 -22885.617} C_VEL
LIN {X 0,Y 171.454,Z 192.129,A -85,B 0,C 180,E1 -22890.597,E2 -22890.597} C_VEL
LIN {X 0,Y 171.395,Z 192.166,A -85,B 0,C 180,E1 -22896.482,E2 -22896.482} C_VEL
LIN {X 0,Y 171.544,Z 193.019,A -85,B 0,C 180,E1 -22897.27,E2 -22897.27} C_VEL
LIN {X 0,Y 173.114,Z 195.954,A -85,B 0,C 180,E1 -22898.226,E2 -22898.226} C_VEL
LIN {X 0,Y 175.086,Z 197.777,A -85,B 0,C 180,E1 -22899.157,E2 -22899.157} C_VEL
LIN {X 0,Y 177.17,Z 201.091,A -85,B 0,C 180,E1 -22900.185,E2 -22900.185} C_VEL
LIN {X 0,Y 178.756,Z 203.013,A -85,B 0,C 180,E1 -22900.901,E2 -22900.901} C_VEL
LIN {X 0,Y 184.501,Z 211.22,A -85,B 0,C 180,E1 -22903.384,E2 -22903.384} C_VEL
LIN {X 0,Y 188.576,Z 217.737,A -85,B 0,C 180,E1 -22905.027,E2 -22905.027} C_VEL
LIN {X 0,Y 194.215,Z 228.709,A -85,B 0,C 180,E1 -22907.216,E2 -22907.216} C_VEL
LIN {X 0,Y 200.403,Z 242.886,A -85,B 0,C 180,E1 -22909.496,E2 -22909.496} C_VEL
LIN {X 0,Y 202.145,Z 247.329,A -85,B 0,C 180,E1 -22910.119,E2 -22910.119} C_VEL
LIN {X 0,Y 199.343,Z 297.302,A -85,B 0,C 180,E1 -22911.806,E2 -22911.806} C_VEL
LIN {X 0,Y 197.588,Z 310.756,A -85,B 0,C 180,E1 -22912.584,E2 -22912.584} C_VEL
LIN {X 0,Y 195.425,Z 323.536,A -85,B 0,C 180,E1 -22913.765,E2 -22913.765} C_VEL
LIN {X 0,Y 192.645,Z 335.341,A -85,B 0,C 180,E1 -22915.25,E2 -22915.25} C_VEL
LIN {X 0,Y 189.459,Z 346.689,A -85,B 0,C 180,E1 -22917.147,E2 -22917.147} C_VEL
LIN {X 0,Y 186.084,Z 356.917,A -85,B 0,C 180,E1 -22919.347,E2 -22919.347} C_VEL
LIN {X 0,Y 182.81,Z 366.098,A -85,B 0,C 180,E1 -22921.906,E2 -22921.906} C_VEL
LIN {X 0,Y 179.275,Z 375.023,A -85,B 0,C 180,E1 -22925.077,E2 -22925.077} C_VEL
LIN {X 0,Y 176.221,Z 382.209,A -85,B 0,C 180,E1 -22928.353,E2 -22928.353} C_VEL
LIN {X 0,Y 173.987,Z 387.055,A -85,B 0,C 180,E1 -22931.148,E2 -22931.148} C_VEL
LIN {X 0,Y 171.986,Z 391.763,A -85,B 0,C 180,E1 -22934.598,E2 -22934.598} C_VEL
LIN {X 0,Y 170.533,Z 395.366,A -85,B 0,C 180,E1 -22938.11,E2 -22938.11} C_VEL
LIN {X 0,Y 169.802,Z 397.227,A -85,B 0,C 180,E1 -22940.472,E2 -22940.472} C_VEL
LIN {X 0,Y 169.349,Z 398.625,A -85,B 0,C 180,E1 -22942.849,E2 -22942.849} C_VEL
LIN {X 0,Y 168.888,Z 400.23,A -85,B 0,C 180,E1 -22947.616,E2 -22947.616} C_VEL
LIN {X 0,Y 168.885,Z 400.459,A -85,B 0,C 180,E1 -22950.001,E2 -22950.001} C_VEL
LIN {X 0,Y 168.893,Z 400.155,A -85,B 0,C 180,E1 -22952.922,E2 -22952.922} C_VEL
LIN {X 0,Y 169.35,Z 398.698,A -85,B 0,C 180,E1 -22957.153,E2 -22957.153} C_VEL
LIN {X 0,Y 169.8,Z 397.332,A -85,B 0,C 180,E1 -22959.531,E2 -22959.531} C_VEL
LIN {X 0,Y 170.957,Z 394.448,A -85,B 0,C 180,E1 -22963.069,E2 -22963.069} C_VEL
LIN {X 0,Y 172.566,Z 390.538,A -85,B 0,C 180,E1 -22966.565,E2 -22966.565} C_VEL
LIN {X 0,Y 174.792,Z 385.495,A -85,B 0,C 180,E1 -22969.985,E2 -22969.985} C_VEL
LIN {X 0,Y 177.637,Z 379.144,A -85,B 0,C 180,E1 -22973.306,E2 -22973.306} C_VEL
LIN {X 0,Y 180.737,Z 371.663,A -85,B 0,C 180,E1 -22976.37,E2 -22976.37} C_VEL
LIN {X 0,Y 183.906,Z 363.109,A -85,B 0,C 180,E1 -22979.16,E2 -22979.16} C_VEL
LIN {X 0,Y 187.454,Z 353.232,A -85,B 0,C 180,E1 -22981.661,E2 -22981.661} C_VEL
LIN {X 0,Y 190.984,Z 342.109,A -85,B 0,C 180,E1 -22983.82,E2 -22983.82} C_VEL
LIN {X 0,Y 193.793,Z 331.209,A -85,B 0,C 180,E1 -22985.468,E2 -22985.468} C_VEL
LIN {X 0,Y 196.385,Z 319.158,A -85,B 0,C 180,E1 -22986.829,E2 -22986.829} C_VEL
LIN {X 0,Y 198.387,Z 306.618,A -85,B 0,C 180,E1 -22987.84,E2 -22987.84} C_VEL
LIN {X 0,Y 199.736,Z 293.882,A -85,B 0,C 180,E1 -22988.485,E2 -22988.485} C_VEL
LIN {X 0,Y 202.213,Z 247.336,A -85,B 0,C 180,E1 -22990.04,E2 -22990.04} C_VEL
LIN {X 0,Y 197.275,Z 235.309,A -85,B 0,C 180,E1 -22991.831,E2 -22991.831} C_VEL
LIN {X 0,Y 192.062,Z 224.204,A -85,B 0,C 180,E1 -22993.802,E2 -22993.802} C_VEL
LIN {X 0,Y 186.556,Z 214.157,A -85,B 0,C 180,E1 -22995.992,E2 -22995.992} C_VEL
LIN {X 0,Y 180.726,Z 205.809,A -85,B 0,C 180,E1 -22998.431,E2 -22998.431} C_VEL
LIN {X 0,Y 177.681,Z 201.58,A -85,B 0,C 180,E1 -22999.811,E2 -22999.811} C_VEL
LIN {X 0,Y 175.369,Z 198.374,A -85,B 0,C 180,E1 -23000.919,E2 -23000.919} C_VEL
LIN {X 0,Y 174.712,Z 197.346,A -85,B 0,C 180,E1 -23001.252,E2 -23001.252} C_VEL
LIN {X 0,Y 172.379,Z 194.953,A -85,B 0,C 180,E1 -23002.39,E2 -23002.39} C_VEL
LIN {X 0,Y 171.494,Z 192.779,A -85,B 0,C 180,E1 -23003.085,E2 -23003.085} C_VEL
LIN {X 0,Y 171.402,Z 192.134,A -85,B 0,C 180,E1 -23003.884,E2 -23003.884} C_VEL
LIN {X 0,Y 171.459,Z 192.126,A -85,B 0,C 180,E1 -23009.404,E2 -23009.404} C_VEL
LIN {X 0,Y 171.459,Z 192.121,A -85,B 0,C 180,E1 -23014.391,E2 -23014.391} C_VEL
LIN {X 0,Y 171.578,Z 192.113,A -85,B 0,C 180,E1 -23020.871,E2 -23020.871} C_VEL
LIN {X 0,Y 171.591,Z 192.092,A -85,B 0,C 180,E1 -23025.774,E2 -23025.774} C_VEL
LIN {X 0,Y 171.873,Z 192.047,A -85,B 0,C 180,E1 -23030.586,E2 -23030.586} C_VEL
LIN {X 0,Y 171.816,Z 192.073,A -85,B 0,C 180,E1 -23035.307,E2 -23035.307} C_VEL
LIN {X 0,Y 172.329,Z 192.009,A -85,B 0,C 180,E1 -23040,E2 -23040} C_VEL
LIN {X 0,Y 171.805,Z 192.057,A -85,B 0,C 180,E1 -23044.693,E2 -23044.693} C_VEL
LIN {X 0,Y 171.843,Z 192.066,A -85,B 0,C 180,E1 -23049.415,E2 -23049.415} C_VEL
LIN {X 0,Y 171.565,Z 192.112,A -85,B 0,C 180,E1 -23054.228,E2 -23054.228} C_VEL
LIN {X 0,Y 171.53,Z 192.104,A -85,B 0,C 180,E1 -23059.548,E2 -23059.548} C_VEL
LIN {X 0,Y 171.458,Z 192.116,A -85,B 0,C 180,E1 -23065.609,E2 -23065.609} C_VEL
LIN {X 0,Y 171.439,Z 192.117,A -85,B 0,C 180,E1 -23070.585,E2 -23070.585} C_VEL
LIN {X 0,Y 171.416,Z 192.235,A -85,B 0,C 180,E1 -23076.385,E2 -23076.385} C_VEL
LIN {X 0,Y 171.637,Z 193.369,A -85,B 0,C 180,E1 -23077.063,E2 -23077.063} C_VEL
LIN {X 0,Y 173.116,Z 195.942,A -85,B 0,C 180,E1 -23077.908,E2 -23077.908} C_VEL
LIN {X 0,Y 175.188,Z 197.944,A -85,B 0,C 180,E1 -23078.897,E2 -23078.897} C_VEL
LIN {X 0,Y 177.103,Z 200.999,A -85,B 0,C 180,E1 -23079.847,E2 -23079.847} C_VEL
LIN {X 0,Y 178.797,Z 203.041,A -85,B 0,C 180,E1 -23080.616,E2 -23080.616} C_VEL
LIN {X 0,Y 182.484,Z 208.886,A -85,B 0,C 180,E1 -23082.281,E2 -23082.281} C_VEL
LIN {X 0,Y 187.422,Z 217.255,A -85,B 0,C 180,E1 -23084.365,E2 -23084.365} C_VEL
LIN {X 0,Y 193.625,Z 229.269,A -85,B 0,C 180,E1 -23086.81,E2 -23086.81} C_VEL
LIN {X 0,Y 199.124,Z 242.014,A -85,B 0,C 180,E1 -23088.876,E2 -23088.876} C_VEL
LIN {X 0,Y 202.096,Z 249.871,A -85,B 0,C 180,E1 -23089.964,E2 -23089.964} C_VEL
LIN {X 0,Y 199.319,Z 300.46,A -85,B 0,C 180,E1 -23091.692,E2 -23091.692} C_VEL
LIN {X 0,Y 197.667,Z 313.595,A -85,B 0,C 180,E1 -23092.469,E2 -23092.469} C_VEL
LIN {X 0,Y 196.54,Z 320.102,A -85,B 0,C 180,E1 -23092.99,E2 -23092.99} C_VEL
LIN {X 0,Y 195.302,Z 323.828,A -85,B 0,C 180,E1 -23093.212,E2 -23093.212} C_VEL
LIN {X 0,Y 191.734,Z 329.582,A -85,B 0,C 180,E1 -23093.32,E2 -23093.32} C_VEL
LIN {X 0,Y 188.022,Z 335.2,A -85,B 0,C 180,E1 -23093.528,E2 -23093.528} C_VEL
LIN {X 0,Y 186.565,Z 338.665,A -85,B 0,C 180,E1 -23093.915,E2 -23093.915} C_VEL
LIN {X 0,Y 183.216,Z 350.045,A -85,B 0,C 180,E1 -23095.875,E2 -23095.875} C_VEL
LIN {X 0,Y 179.614,Z 360.174,A -85,B 0,C 180,E1 -23098.114,E2 -23098.114} C_VEL
LIN {X 0,Y 176.017,Z 369.3,A -85,B 0,C 180,E1 -23100.717,E2 -23100.717} C_VEL
LIN {X 0,Y 172.67,Z 377.591,A -85,B 0,C 180,E1 -23103.762,E2 -23103.762} C_VEL
LIN {X 0,Y 169.231,Z 385.35,A -85,B 0,C 180,E1 -23107.409,E2 -23107.409} C_VEL
LIN {X 0,Y 166.081,Z 391.862,A -85,B 0,C 180,E1 -23111.495,E2 -23111.495} C_VEL
LIN {X 0,Y 164.189,Z 396.172,A -85,B 0,C 180,E1 -23115.117,E2 -23115.117} C_VEL
LIN {X 0,Y 163.228,Z 398.453,A -85,B 0,C 180,E1 -23117.567,E2 -23117.567} C_VEL
LIN {X 0,Y 162.545,Z 400.3,A -85,B 0,C 180,E1 -23120.04,E2 -23120.04} C_VEL
LIN {X 0,Y 162.125,Z 401.684,A -85,B 0,C 180,E1 -23122.527,E2 -23122.527} C_VEL
LIN {X 0,Y 161.857,Z 402.673,A -85,B 0,C 180,E1 -23125.017,E2 -23125.017} C_VEL
LIN {X 0,Y 161.709,Z 403.387,A -85,B 0,C 180,E1 -23128.377,E2 -23128.377} C_VEL
LIN {X 0,Y 161.725,Z 403.371,A -85,B 0,C 180,E1 -23131.805,E2 -23131.805} C_VEL
LIN {X 0,Y 161.857,Z 402.649,A -85,B 0,C 180,E1 -23134.981,E2 -23134.981} C_VEL
LIN {X 0,Y 162.125,Z 401.652,A -85,B 0,C 180,E1 -23137.471,E2 -23137.471} C_VEL
LIN {X 0,Y 162.547,Z 400.253,A -85,B 0,C 180,E1 -23139.958,E2 -23139.958} C_VEL
LIN {X 0,Y 163.694,Z 397.32,A -85,B 0,C 180,E1 -23143.657,E2 -23143.657} C_VEL
LIN {X 0,Y 165.331,Z 393.351,A -85,B 0,C 180,E1 -23147.31,E2 -23147.31} C_VEL
LIN {X 0,Y 168.245,Z 387.248,A -85,B 0,C 180,E1 -23151.437,E2 -23151.437} C_VEL
LIN {X 0,Y 171.277,Z 380.626,A -85,B 0,C 180,E1 -23154.847,E2 -23154.847} C_VEL
LIN {X 0,Y 174.664,Z 372.459,A -85,B 0,C 180,E1 -23158.148,E2 -23158.148} C_VEL
LIN {X 0,Y 178.089,Z 363.823,A -85,B 0,C 180,E1 -23160.864,E2 -23160.864} C_VEL
LIN {X 0,Y 181.887,Z 353.334,A -85,B 0,C 180,E1 -23163.407,E2 -23163.407} C_VEL
LIN {X 0,Y 185.216,Z 342.952,A -85,B 0,C 180,E1 -23165.354,E2 -23165.354} C_VEL
LIN {X 0,Y 188.318,Z 331.557,A -85,B 0,C 180,E1 -23166.995,E2 -23166.995} C_VEL
LIN {X 0,Y 190.789,Z 319.807,A -85,B 0,C 180,E1 -23168.264,E2 -23168.264} C_VEL
LIN {X 0,Y 192.948,Z 306.572,A -85,B 0,C 180,E1 -23169.23,E2 -23169.23} C_VEL
LIN {X 0,Y 194.17,Z 293.462,A -85,B 0,C 180,E1 -23169.845,E2 -23169.845} C_VEL
LIN {X 0,Y 196.538,Z 251.875,A -85,B 0,C 180,E1 -23171.222,E2 -23171.222} C_VEL
LIN {X 0,Y 190.495,Z 236.686,A -85,B 0,C 180,E1 -23173.598,E2 -23173.598} C_VEL
LIN {X 0,Y 184.922,Z 225.008,A -85,B 0,C 180,E1 -23175.894,E2 -23175.894} C_VEL
LIN {X 0,Y 179.281,Z 214.899,A -85,B 0,C 180,E1 -23178.374,E2 -23178.374} C_VEL
LIN {X 0,Y 174.536,Z 207.399,A -85,B 0,C 180,E1 -23180.626,E2 -23180.626} C_VEL
LIN {X 0,Y 171.857,Z 203.609,A -85,B 0,C 180,E1 -23181.974,E2 -23181.974} C_VEL
LIN {X 0,Y 168.875,Z 200.001,A -85,B 0,C 180,E1 -23183.535,E2 -23183.535} C_VEL
LIN {X 0,Y 167.879,Z 198.257,A -85,B 0,C 180,E1 -23184.12,E2 -23184.12} C_VEL
LIN {X 0,Y 165.589,Z 196.155,A -85,B 0,C 180,E1 -23185.383,E2 -23185.383} C_VEL
LIN {X 0,Y 164.478,Z 193.757,A -85,B 0,C 180,E1 -23186.256,E2 -23186.256} C_VEL
LIN {X 0,Y 164.348,Z 193.044,A -85,B 0,C 180,E1 -23187.1,E2 -23187.1} C_VEL
LIN {X 0,Y 164.333,Z 193.003,A -85,B 0,C 180,E1 -23191.937,E2 -23191.937} C_VEL
LIN {X 0,Y 164.4,Z 192.991,A -85,B 0,C 180,E1 -23194.691,E2 -23194.691} C_VEL
LIN {X 0,Y 164.457,Z 192.988,A -85,B 0,C 180,E1 -23200.072,E2 -23200.072} C_VEL
LIN {X 0,Y 164.511,Z 192.994,A -85,B 0,C 180,E1 -23205.148,E2 -23205.148} C_VEL
LIN {X 0,Y 164.795,Z 192.939,A -85,B 0,C 180,E1 -23210.178,E2 -23210.178} C_VEL
LIN {X 0,Y 164.842,Z 192.946,A -85,B 0,C 180,E1 -23212.652,E2 -23212.652} C_VEL
LIN {X 0,Y 165.039,Z 192.914,A -85,B 0,C 180,E1 -23217.559,E2 -23217.559} C_VEL
LIN {X 0,Y 165.287,Z 192.885,A -85,B 0,C 180,E1 -23220,E2 -23220} C_VEL
LIN {X 0,Y 164.761,Z 192.952,A -85,B 0,C 180,E1 -23224.894,E2 -23224.894} C_VEL
LIN {X 0,Y 164.839,Z 192.934,A -85,B 0,C 180,E1 -23227.349,E2 -23227.349} C_VEL
LIN {X 0,Y 164.745,Z 192.946,A -85,B 0,C 180,E1 -23231.146,E2 -23231.146} C_VEL
LIN {X 0,Y 164.492,Z 192.977,A -85,B 0,C 180,E1 -23237.402,E2 -23237.402} C_VEL
LIN {X 0,Y 164.47,Z 192.989,A -85,B 0,C 180,E1 -23239.99,E2 -23239.99} C_VEL
LIN {X 0,Y 164.388,Z 192.997,A -85,B 0,C 180,E1 -23246.135,E2 -23246.135} C_VEL
LIN {X 0,Y 164.382,Z 192.968,A -85,B 0,C 180,E1 -23252.38,E2 -23252.38} C_VEL
LIN {X 0,Y 164.372,Z 193.328,A -85,B 0,C 180,E1 -23253.594,E2 -23253.594} C_VEL
LIN {X 0,Y 164.723,Z 194.518,A -85,B 0,C 180,E1 -23254.204,E2 -23254.204} C_VEL
LIN {X 0,Y 166.506,Z 197.254,A -85,B 0,C 180,E1 -23255.324,E2 -23255.324} C_VEL
LIN {X 0,Y 168.351,Z 198.877,A -85,B 0,C 180,E1 -23256.319,E2 -23256.319} C_VEL
LIN {X 0,Y 170.401,Z 202.124,A -85,B 0,C 180,E1 -23257.47,E2 -23257.47} C_VEL
LIN {X 0,Y 172.054,Z 203.957,A -85,B 0,C 180,E1 -23258.306,E2 -23258.306} C_VEL
LIN {X 0,Y 174.799,Z 207.696,A -85,B 0,C 180,E1 -23259.671,E2 -23259.671} C_VEL
LIN {X 0,Y 180.825,Z 216.515,A -85,B 0,C 180,E1 -23262.44,E2 -23262.44} C_VEL
LIN {X 0,Y 184.778,Z 223.083,A -85,B 0,C 180,E1 -23264.128,E2 -23264.128} C_VEL
LIN {X 0,Y 189.898,Z 233.339,A -85,B 0,C 180,E1 -23266.233,E2 -23266.233} C_VEL
LIN {X 0,Y 195.515,Z 246.459,A -85,B 0,C 180,E1 -23268.429,E2 -23268.429} C_VEL
LIN {X 0,Y 196.64,Z 249.438,A -85,B 0,C 180,E1 -23268.862,E2 -23268.862} C_VEL
LIN {X 0,Y 193.862,Z 297.04,A -85,B 0,C 180,E1 -23270.495,E2 -23270.495} C_VEL
LIN {X 0,Y 192.046,Z 310.466,A -85,B 0,C 180,E1 -23271.268,E2 -23271.268} C_VEL
LIN {X 0,Y 189.982,Z 322.526,A -85,B 0,C 180,E1 -23272.385,E2 -23272.385} C_VEL
LIN {X 0,Y 187.303,Z 333.828,A -85,B 0,C 180,E1 -23273.776,E2 -23273.776} C_VEL
LIN {X 0,Y 183.961,Z 345.468,A -85,B 0,C 180,E1 -23275.703,E2 -23275.703} C_VEL
LIN {X 0,Y 180.392,Z 355.928,A -85,B 0,C 180,E1 -23277.941,E2 -23277.941} C_VEL
LIN {X 0,Y 177.197,Z 364.475,A -85,B 0,C 180,E1 -23280.281,E2 -23280.281} C_VEL
LIN {X 0,Y 174.053,Z 372.431,A -85,B 0,C 180,E1 -23283.02,E2 -23283.02} C_VEL
LIN {X 0,Y 170.688,Z 380.048,A -85,B 0,C 180,E1 -23286.333,E2 -23286.333} C_VEL
LIN {X 0,Y 167.27,Z 387.121,A -85,B 0,C 180,E1 -23290.361,E2 -23290.361} C_VEL
LIN {X 0,Y 165.134,Z 391.83,A -85,B 0,C 180,E1 -23293.942,E2 -23293.942} C_VEL
LIN {X 0,Y 163.566,Z 395.432,A -85,B 0,C 180,E1 -23297.595,E2 -23297.595} C_VEL
LIN {X 0,Y 162.788,Z 397.293,A -85,B 0,C 180,E1 -23300.057,E2 -23300.057} C_VEL
LIN {X 0,Y 162.298,Z 398.69,A -85,B 0,C 180,E1 -23302.537,E2 -23302.537} C_VEL
LIN {X 0,Y 161.798,Z 400.295,A -85,B 0,C 180,E1 -23307.512,E2 -23307.512} C_VEL
LIN {X 0,Y 161.802,Z 400.523,A -85,B 0,C 180,E1 -23310.001,E2 -23310.001} C_VEL
LIN {X 0,Y 161.798,Z 400.327,A -85,B 0,C 180,E1 -23312.491,E2 -23312.491} C_VEL
LIN {X 0,Y 162.298,Z 398.763,A -85,B 0,C 180,E1 -23317.465,E2 -23317.465} C_VEL
LIN {X 0,Y 162.788,Z 397.397,A -85,B 0,C 180,E1 -23319.945,E2 -23319.945} C_VEL
LIN {X 0,Y 164.019,Z 394.512,A -85,B 0,C 180,E1 -23323.632,E2 -23323.632} C_VEL
LIN {X 0,Y 165.74,Z 390.602,A -85,B 0,C 180,E1 -23327.268,E2 -23327.268} C_VEL
LIN {X 0,Y 168.135,Z 385.558,A -85,B 0,C 180,E1 -23330.812,E2 -23330.812} C_VEL
LIN {X 0,Y 171.119,Z 379.207,A -85,B 0,C 180,E1 -23334.25,E2 -23334.25} C_VEL
LIN {X 0,Y 174.76,Z 370.734,A -85,B 0,C 180,E1 -23337.78,E2 -23337.78} C_VEL
LIN {X 0,Y 178.421,Z 361.39,A -85,B 0,C 180,E1 -23340.802,E2 -23340.802} C_VEL
LIN {X 0,Y 182.257,Z 351.016,A -85,B 0,C 180,E1 -23343.332,E2 -23343.332} C_VEL
LIN {X 0,Y 185.97,Z 339.32,A -85,B 0,C 180,E1 -23345.524,E2 -23345.524} C_VEL
LIN {X 0,Y 188.976,Z 327.647,A -85,B 0,C 180,E1 -23347.181,E2 -23347.181} C_VEL
LIN {X 0,Y 191.42,Z 315.502,A -85,B 0,C 180,E1 -23348.452,E2 -23348.452} C_VEL
LIN {X 0,Y 193.434,Z 302.139,A -85,B 0,C 180,E1 -23349.404,E2 -23349.404} C_VEL
LIN {X 0,Y 194.482,Z 288.742,A -85,B 0,C 180,E1 -23349.999,E2 -23349.999} C_VEL
LIN {X 0,Y 196.717,Z 249.435,A -85,B 0,C 180,E1 -23351.3,E2 -23351.3} C_VEL
LIN {X 0,Y 191.064,Z 235.692,A -85,B 0,C 180,E1 -23353.504,E2 -23353.504} C_VEL
LIN {X 0,Y 186.031,Z 225.293,A -85,B 0,C 180,E1 -23355.555,E2 -23355.555} C_VEL
LIN {X 0,Y 181.758,Z 217.899,A -85,B 0,C 180,E1 -23357.369,E2 -23357.369} C_VEL
LIN {X 0,Y 177.025,Z 210.945,A -85,B 0,C 180,E1 -23359.487,E2 -23359.487} C_VEL
LIN {X 0,Y 174.025,Z 206.788,A -85,B 0,C 180,E1 -23360.924,E2 -23360.924} C_VEL
LIN {X 0,Y 171.45,Z 203.133,A -85,B 0,C 180,E1 -23362.243,E2 -23362.243} C_VEL
LIN {X 0,Y 168.854,Z 199.925,A -85,B 0,C 180,E1 -23363.622,E2 -23363.622} C_VEL
LIN {X 0,Y 167.978,Z 198.329,A -85,B 0,C 180,E1 -23364.144,E2 -23364.144} C_VEL
LIN {X 0,Y 165.574,Z 196.161,A -85,B 0,C 180,E1 -23365.476,E2 -23365.476} C_VEL
LIN {X 0,Y 164.445,Z 193.656,A -85,B 0,C 180,E1 -23366.423,E2 -23366.423} C_VEL
LIN {X 0,Y 164.371,Z 193.019,A -85,B 0,C 180,E1 -23367.273,E2 -23367.273} C_VEL
LIN {X 0,Y 164.34,Z 192.995,A -85,B 0,C 180,E1 -23371.938,E2 -23371.938} C_VEL
LIN {X 0,Y 164.407,Z 193.003,A -85,B 0,C 180,E1 -23374.692,E2 -23374.692} C_VEL
LIN {X 0,Y 164.485,Z 192.986,A -85,B 0,C 180,E1 -23380.051,E2 -23380.051} C_VEL
LIN {X 0,Y 164.533,Z 192.966,A -85,B 0,C 180,E1 -23385.15,E2 -23385.15} C_VEL
LIN {X 0,Y 164.797,Z 192.929,A -85,B 0,C 180,E1 -23390.178,E2 -23390.178} C_VEL
LIN {X 0,Y 164.845,Z 192.932,A -85,B 0,C 180,E1 -23392.651,E2 -23392.651} C_VEL
LIN {X 0,Y 165.046,Z 192.898,A -85,B 0,C 180,E1 -23397.559,E2 -23397.559} C_VEL
LIN {X 0,Y 165.291,Z 192.884,A -85,B 0,C 180,E1 -23400,E2 -23400} C_VEL
LIN {X 0,Y 164.753,Z 192.935,A -85,B 0,C 180,E1 -23404.894,E2 -23404.894} C_VEL
LIN {X 0,Y 164.824,Z 192.949,A -85,B 0,C 180,E1 -23407.349,E2 -23407.349} C_VEL
LIN {X 0,Y 164.701,Z 192.943,A -85,B 0,C 180,E1 -23411.058,E2 -23411.058} C_VEL
LIN {X 0,Y 164.469,Z 192.975,A -85,B 0,C 180,E1 -23417.405,E2 -23417.405} C_VEL
LIN {X 0,Y 164.472,Z 192.988,A -85,B 0,C 180,E1 -23419.989,E2 -23419.989} C_VEL
LIN {X 0,Y 164.385,Z 193.003,A -85,B 0,C 180,E1 -23426.128,E2 -23426.128} C_VEL
LIN {X 0,Y 164.378,Z 193.028,A -85,B 0,C 180,E1 -23432.374,E2 -23432.374} C_VEL
LIN {X 0,Y 164.41,Z 193.55,A -85,B 0,C 180,E1 -23433.409,E2 -23433.409} C_VEL
LIN {X 0,Y 165.304,Z 195.789,A -85,B 0,C 180,E1 -23434.276,E2 -23434.276} C_VEL
LIN {X 0,Y 167.664,Z 198.141,A -85,B 0,C 180,E1 -23435.61,E2 -23435.61} C_VEL
LIN {X 0,Y 168.301,Z 198.838,A -85,B 0,C 180,E1 -23435.961,E2 -23435.961} C_VEL
LIN {X 0,Y 170.344,Z 202.016,A -85,B 0,C 180,E1 -23437.113,E2 -23437.113} C_VEL
LIN {X 0,Y 172.043,Z 203.878,A -85,B 0,C 180,E1 -23437.978,E2 -23437.978} C_VEL
LIN {X 0,Y 174.722,Z 207.597,A -85,B 0,C 180,E1 -23439.324,E2 -23439.324} C_VEL
LIN {X 0,Y 179.007,Z 214.447,A -85,B 0,C 180,E1 -23441.376,E2 -23441.376} C_VEL
LIN {X 0,Y 183.181,Z 221.623,A -85,B 0,C 180,E1 -23443.239,E2 -23443.239} C_VEL
LIN {X 0,Y 189.307,Z 233.767,A -85,B 0,C 180,E1 -23445.805,E2 -23445.805} C_VEL
LIN {X 0,Y 194.688,Z 246.685,A -85,B 0,C 180,E1 -23447.955,E2 -23447.955} C_VEL
LIN {X 0,Y 196.535,Z 251.61,A -85,B 0,C 180,E1 -23448.673,E2 -23448.673} C_VEL
LIN {X 0,Y 193.993,Z 298.151,A -85,B 0,C 180,E1 -23450.283,E2 -23450.283} C_VEL
LIN {X 0,Y 192.461,Z 311.13,A -85,B 0,C 180,E1 -23451.003,E2 -23451.003} C_VEL
LIN {X 0,Y 190.108,Z 323.915,A -85,B 0,C 180,E1 -23452.077,E2 -23452.077} C_VEL
LIN {X 0,Y 187.357,Z 335.55,A -85,B 0,C 180,E1 -23453.452,E2 -23453.452} C_VEL
LIN {X 0,Y 186.565,Z 338.665,A -85,B 0,C 180,E1 -23453.915,E2 -23453.915} C_VEL
LIN {X 0,Y 184.611,Z 343.815,A -85,B 0,C 180,E1 -23454.621,E2 -23454.621} C_VEL
LIN {X 0,Y 179.661,Z 351.853,A -85,B 0,C 180,E1 -23455.615,E2 -23455.615} C_VEL
LIN {X 0,Y 174.478,Z 359.406,A -85,B 0,C 180,E1 -23456.817,E2 -23456.817} C_VEL
LIN {X 0,Y 172.154,Z 363.763,A -85,B 0,C 180,E1 -23457.861,E2 -23457.861} C_VEL
LIN {X 0,Y 168.493,Z 372.438,A -85,B 0,C 180,E1 -23460.652,E2 -23460.652} C_VEL
LIN {X 0,Y 164.805,Z 380.847,A -85,B 0,C 180,E1 -23464.174,E2 -23464.174} C_VEL
LIN {X 0,Y 161.653,Z 387.313,A -85,B 0,C 180,E1 -23467.64,E2 -23467.64} C_VEL
LIN {X 0,Y 158.542,Z 393.379,A -85,B 0,C 180,E1 -23471.922,E2 -23471.922} C_VEL
LIN {X 0,Y 156.777,Z 397.323,A -85,B 0,C 180,E1 -23475.725,E2 -23475.725} C_VEL
LIN {X 0,Y 155.531,Z 400.235,A -85,B 0,C 180,E1 -23479.586,E2 -23479.586} C_VEL
LIN {X 0,Y 155.059,Z 401.62,A -85,B 0,C 180,E1 -23482.184,E2 -23482.184} C_VEL
LIN {X 0,Y 154.769,Z 402.608,A -85,B 0,C 180,E1 -23484.788,E2 -23484.788} C_VEL
LIN {X 0,Y 154.633,Z 403.375,A -85,B 0,C 180,E1 -23489.149,E2 -23489.149} C_VEL
LIN {X 0,Y 154.633,Z 403.195,A -85,B 0,C 180,E1 -23492.604,E2 -23492.604} C_VEL
LIN {X 0,Y 154.768,Z 402.584,A -85,B 0,C 180,E1 -23495.21,E2 -23495.21} C_VEL
LIN {X 0,Y 155.059,Z 401.587,A -85,B 0,C 180,E1 -23497.814,E2 -23497.814} C_VEL
LIN {X 0,Y 155.532,Z 400.187,A -85,B 0,C 180,E1 -23500.412,E2 -23500.412} C_VEL
LIN {X 0,Y 156.777,Z 397.254,A -85,B 0,C 180,E1 -23504.272,E2 -23504.272} C_VEL
LIN {X 0,Y 158.538,Z 393.285,A -85,B 0,C 180,E1 -23508.076,E2 -23508.076} C_VEL
LIN {X 0,Y 161.645,Z 387.182,A -85,B 0,C 180,E1 -23512.359,E2 -23512.359} C_VEL
LIN {X 0,Y 164.799,Z 380.687,A -85,B 0,C 180,E1 -23515.824,E2 -23515.824} C_VEL
LIN {X 0,Y 168.477,Z 372.243,A -85,B 0,C 180,E1 -23519.348,E2 -23519.348} C_VEL
LIN {X 0,Y 172.033,Z 363.755,A -85,B 0,C 180,E1 -23522.077,E2 -23522.077} C_VEL
LIN {X 0,Y 176.001,Z 353.266,A -85,B 0,C 180,E1 -23524.68,E2 -23524.68} C_VEL
LIN {X 0,Y 179.483,Z 342.883,A -85,B 0,C 180,E1 -23526.663,E2 -23526.663} C_VEL
LIN {X 0,Y 182.7,Z 331.486,A -85,B 0,C 180,E1 -23528.335,E2 -23528.335} C_VEL
LIN {X 0,Y 185.27,Z 319.734,A -85,B 0,C 180,E1 -23529.623,E2 -23529.623} C_VEL
LIN {X 0,Y 187.496,Z 306.598,A -85,B 0,C 180,E1 -23530.594,E2 -23530.594} C_VEL
LIN {X 0,Y 188.788,Z 293.336,A -85,B 0,C 180,E1 -23531.225,E2 -23531.225} C_VEL
LIN {X 0,Y 191.077,Z 253.742,A -85,B 0,C 180,E1 -23532.575,E2 -23532.575} C_VEL
LIN {X 0,Y 185.623,Z 239.88,A -85,B 0,C 180,E1 -23534.872,E2 -23534.872} C_VEL
LIN {X 0,Y 180.145,Z 228.344,A -85,B 0,C 180,E1 -23537.288,E2 -23537.288} C_VEL
LIN {X 0,Y 174.234,Z 217.588,A -85,B 0,C 180,E1 -23540.102,E2 -23540.102} C_VEL
LIN {X 0,Y 170.98,Z 212.697,A -85,B 0,C 180,E1 -23541.744,E2 -23541.744} C_VEL
LIN {X 0,Y 167.91,Z 208.46,A -85,B 0,C 180,E1 -23543.384,E2 -23543.384} C_VEL
LIN {X 0,Y 165.29,Z 204.712,A -85,B 0,C 180,E1 -23544.896,E2 -23544.896} C_VEL
LIN {X 0,Y 162.316,Z 201.344,A -85,B 0,C 180,E1 -23546.678,E2 -23546.678} C_VEL
LIN {X 0,Y 161.09,Z 199.314,A -85,B 0,C 180,E1 -23547.509,E2 -23547.509} C_VEL
LIN {X 0,Y 158.767,Z 197.349,A -85,B 0,C 180,E1 -23549.014,E2 -23549.014} C_VEL
LIN {X 0,Y 157.419,Z 194.671,A -85,B 0,C 180,E1 -23550.22,E2 -23550.22} C_VEL
LIN {X 0,Y 157.285,Z 193.922,A -85,B 0,C 180,E1 -23551.293,E2 -23551.293} C_VEL
LIN {X 0,Y 157.297,Z 193.87,A -85,B 0,C 180,E1 -23556.289,E2 -23556.289} C_VEL
LIN {X 0,Y 157.386,Z 193.873,A -85,B 0,C 180,E1 -23559.67,E2 -23559.67} C_VEL
LIN {X 0,Y 157.44,Z 193.866,A -85,B 0,C 180,E1 -23564.465,E2 -23564.465} C_VEL
LIN {X 0,Y 157.719,Z 193.816,A -85,B 0,C 180,E1 -23569.733,E2 -23569.733} C_VEL
LIN {X 0,Y 157.8,Z 193.827,A -85,B 0,C 180,E1 -23572.322,E2 -23572.322} C_VEL
LIN {X 0,Y 158.25,Z 193.761,A -85,B 0,C 180,E1 -23580,E2 -23580} C_VEL
LIN {X 0,Y 157.777,Z 193.809,A -85,B 0,C 180,E1 -23587.68,E2 -23587.68} C_VEL
LIN {X 0,Y 157.674,Z 193.828,A -85,B 0,C 180,E1 -23591.315,E2 -23591.315} C_VEL
LIN {X 0,Y 157.462,Z 193.844,A -85,B 0,C 180,E1 -23595.533,E2 -23595.533} C_VEL
LIN {X 0,Y 157.366,Z 193.864,A -85,B 0,C 180,E1 -23600.934,E2 -23600.934} C_VEL
LIN {X 0,Y 157.309,Z 193.874,A -85,B 0,C 180,E1 -23606.685,E2 -23606.685} C_VEL
LIN {X 0,Y 157.328,Z 194.154,A -85,B 0,C 180,E1 -23609.523,E2 -23609.523} C_VEL
LIN {X 0,Y 157.672,Z 195.317,A -85,B 0,C 180,E1 -23610.281,E2 -23610.281} C_VEL
LIN {X 0,Y 159.203,Z 197.847,A -85,B 0,C 180,E1 -23611.461,E2 -23611.461} C_VEL
LIN {X 0,Y 161.529,Z 199.815,A -85,B 0,C 180,E1 -23612.948,E2 -23612.948} C_VEL
LIN {X 0,Y 163.801,Z 203.285,A -85,B 0,C 180,E1 -23614.424,E2 -23614.424} C_VEL
LIN {X 0,Y 165.406,Z 204.914,A -85,B 0,C 180,E1 -23615.349,E2 -23615.349} C_VEL
LIN {X 0,Y 168.164,Z 208.743,A -85,B 0,C 180,E1 -23616.925,E2 -23616.925} C_VEL
LIN {X 0,Y 172.875,Z 215.436,A -85,B 0,C 180,E1 -23619.394,E2 -23619.394} C_VEL
LIN {X 0,Y 177.22,Z 221.815,A -85,B 0,C 180,E1 -23621.464,E2 -23621.464} C_VEL
LIN {X 0,Y 181.14,Z 228.597,A -85,B 0,C 180,E1 -23623.239,E2 -23623.239} C_VEL
LIN {X 0,Y 185.761,Z 238.187,A -85,B 0,C 180,E1 -23625.253,E2 -23625.253} C_VEL
LIN {X 0,Y 190.935,Z 250.685,A -85,B 0,C 180,E1 -23627.406,E2 -23627.406} C_VEL
LIN {X 0,Y 191.237,Z 252.049,A -85,B 0,C 180,E1 -23627.558,E2 -23627.558} C_VEL
LIN {X 0,Y 188.37,Z 297.654,A -85,B 0,C 180,E1 -23629.145,E2 -23629.145} C_VEL
LIN {X 0,Y 186.493,Z 311.131,A -85,B 0,C 180,E1 -23629.955,E2 -23629.955} C_VEL
LIN {X 0,Y 184.195,Z 323.679,A -85,B 0,C 180,E1 -23631.16,E2 -23631.16} C_VEL
LIN {X 0,Y 181.181,Z 335.481,A -85,B 0,C 180,E1 -23632.695,E2 -23632.695} C_VEL
LIN {X 0,Y 177.702,Z 346.827,A -85,B 0,C 180,E1 -23634.663,E2 -23634.663} C_VEL
LIN {X 0,Y 174.02,Z 357.053,A -85,B 0,C 180,E1 -23636.963,E2 -23636.963} C_VEL
LIN {X 0,Y 170.38,Z 366.233,A -85,B 0,C 180,E1 -23639.651,E2 -23639.651} C_VEL
LIN {X 0,Y 166.498,Z 375.157,A -85,B 0,C 180,E1 -23643.016,E2 -23643.016} C_VEL
LIN {X 0,Y 163.088,Z 382.342,A -85,B 0,C 180,E1 -23646.51,E2 -23646.51} C_VEL
LIN {X 0,Y 160.594,Z 387.188,A -85,B 0,C 180,E1 -23649.508,E2 -23649.508} C_VEL
LIN {X 0,Y 158.309,Z 391.896,A -85,B 0,C 180,E1 -23653.23,E2 -23653.23} C_VEL
LIN {X 0,Y 156.624,Z 395.498,A -85,B 0,C 180,E1 -23657.036,E2 -23657.036} C_VEL
LIN {X 0,Y 155.797,Z 397.358,A -85,B 0,C 180,E1 -23659.606,E2 -23659.606} C_VEL
LIN {X 0,Y 155.242,Z 398.756,A -85,B 0,C 180,E1 -23662.196,E2 -23662.196} C_VEL
LIN {X 0,Y 154.701,Z 400.36,A -85,B 0,C 180,E1 -23667.397,E2 -23667.397} C_VEL
LIN {X 0,Y 154.677,Z 400.504,A -85,B 0,C 180,E1 -23671.597,E2 -23671.597} C_VEL
LIN {X 0,Y 154.871,Z 399.801,A -85,B 0,C 180,E1 -23675.208,E2 -23675.208} C_VEL
LIN {X 0,Y 155.242,Z 398.827,A -85,B 0,C 180,E1 -23677.807,E2 -23677.807} C_VEL
LIN {X 0,Y 155.796,Z 397.461,A -85,B 0,C 180,E1 -23680.396,E2 -23680.396} C_VEL
LIN {X 0,Y 157.098,Z 394.576,A -85,B 0,C 180,E1 -23684.245,E2 -23684.245} C_VEL
LIN {X 0,Y 158.942,Z 390.666,A -85,B 0,C 180,E1 -23688.031,E2 -23688.031} C_VEL
LIN {X 0,Y 161.517,Z 385.622,A -85,B 0,C 180,E1 -23691.707,E2 -23691.707} C_VEL
LIN {X 0,Y 164.649,Z 379.271,A -85,B 0,C 180,E1 -23695.268,E2 -23695.268} C_VEL
LIN {X 0,Y 168.226,Z 371.406,A -85,B 0,C 180,E1 -23698.679,E2 -23698.679} C_VEL
LIN {X 0,Y 171.622,Z 363.233,A -85,B 0,C 180,E1 -23701.475,E2 -23701.475} C_VEL
LIN {X 0,Y 175.542,Z 353.354,A -85,B 0,C 180,E1 -23704.091,E2 -23704.091} C_VEL
LIN {X 0,Y 179.367,Z 342.23,A -85,B 0,C 180,E1 -23706.344,E2 -23706.344} C_VEL
LIN {X 0,Y 182.413,Z 331.327,A -85,B 0,C 180,E1 -23708.057,E2 -23708.057} C_VEL
LIN {X 0,Y 185.225,Z 319.273,A -85,B 0,C 180,E1 -23709.461,E2 -23709.461} C_VEL
LIN {X 0,Y 187.418,Z 306.532,A -85,B 0,C 180,E1 -23710.512,E2 -23710.512} C_VEL
LIN {X 0,Y 188.861,Z 293.594,A -85,B 0,C 180,E1 -23711.18,E2 -23711.18} C_VEL
LIN {X 0,Y 191.327,Z 251.483,A -85,B 0,C 180,E1 -23712.634,E2 -23712.634} C_VEL
LIN {X 0,Y 185.601,Z 237.641,A -85,B 0,C 180,E1 -23715.024,E2 -23715.024} C_VEL
LIN {X 0,Y 180.238,Z 226.722,A -85,B 0,C 180,E1 -23717.386,E2 -23717.386} C_VEL
LIN {X 0,Y 176.022,Z 219.911,A -85,B 0,C 180,E1 -23719.318,E2 -23719.318} C_VEL
LIN {X 0,Y 170.821,Z 212.41,A -85,B 0,C 180,E1 -23721.892,E2 -23721.892} C_VEL
LIN {X 0,Y 168.121,Z 208.681,A -85,B 0,C 180,E1 -23723.344,E2 -23723.344} C_VEL
LIN {X 0,Y 165.403,Z 204.857,A -85,B 0,C 180,E1 -23724.913,E2 -23724.913} C_VEL
LIN {X 0,Y 162.325,Z 201.318,A -85,B 0,C 180,E1 -23726.772,E2 -23726.772} C_VEL
LIN {X 0,Y 161.219,Z 199.349,A -85,B 0,C 180,E1 -23727.538,E2 -23727.538} C_VEL
LIN {X 0,Y 158.798,Z 197.35,A -85,B 0,C 180,E1 -23729.113,E2 -23729.113} C_VEL
LIN {X 0,Y 157.386,Z 194.451,A -85,B 0,C 180,E1 -23730.489,E2 -23730.489} C_VEL
LIN {X 0,Y 157.295,Z 193.927,A -85,B 0,C 180,E1 -23731.295,E2 -23731.295} C_VEL
LIN {X 0,Y 157.304,Z 193.877,A -85,B 0,C 180,E1 -23736.29,E2 -23736.29} C_VEL
LIN {X 0,Y 157.409,Z 193.87,A -85,B 0,C 180,E1 -23741.788,E2 -23741.788} C_VEL
LIN {X 0,Y 157.547,Z 193.857,A -85,B 0,C 180,E1 -23747.112,E2 -23747.112} C_VEL
LIN {X 0,Y 157.726,Z 193.812,A -85,B 0,C 180,E1 -23749.733,E2 -23749.733} C_VEL
LIN {X 0,Y 157.783,Z 193.808,A -85,B 0,C 180,E1 -23752.321,E2 -23752.321} C_VEL
LIN {X 0,Y 158.254,Z 193.76,A -85,B 0,C 180,E1 -23760,E2 -23760} C_VEL
LIN {X 0,Y 157.761,Z 193.832,A -85,B 0,C 180,E1 -23767.68,E2 -23767.68} C_VEL
LIN {X 0,Y 157.632,Z 193.823,A -85,B 0,C 180,E1 -23771.227,E2 -23771.227} C_VEL
LIN {X 0,Y 157.432,Z 193.866,A -85,B 0,C 180,E1 -23775.536,E2 -23775.536} C_VEL
LIN {X 0,Y 157.366,Z 193.884,A -85,B 0,C 180,E1 -23780.933,E2 -23780.933} C_VEL
LIN {X 0,Y 157.31,Z 193.892,A -85,B 0,C 180,E1 -23786.681,E2 -23786.681} C_VEL
LIN {X 0,Y 157.314,Z 194.122,A -85,B 0,C 180,E1 -23789.067,E2 -23789.067} C_VEL
LIN {X 0,Y 157.598,Z 195.199,A -85,B 0,C 180,E1 -23789.835,E2 -23789.835} C_VEL
LIN {X 0,Y 159.092,Z 197.716,A -85,B 0,C 180,E1 -23791.012,E2 -23791.012} C_VEL
LIN {X 0,Y 161.518,Z 199.777,A -85,B 0,C 180,E1 -23792.579,E2 -23792.579} C_VEL
LIN {X 0,Y 163.484,Z 202.921,A -85,B 0,C 180,E1 -23793.884,E2 -23793.884} C_VEL
LIN {X 0,Y 165.499,Z 205.017,A -85,B 0,C 180,E1 -23795.063,E2 -23795.063} C_VEL
LIN {X 0,Y 167.99,Z 208.536,A -85,B 0,C 180,E1 -23796.502,E2 -23796.502} C_VEL
LIN {X 0,Y 169.157,Z 210.077,A -85,B 0,C 180,E1 -23797.138,E2 -23797.138} C_VEL
LIN {X 0,Y 172.793,Z 215.264,A -85,B 0,C 180,E1 -23799.036,E2 -23799.036} C_VEL
LIN {X 0,Y 178.057,Z 224.296,A -85,B 0,C 180,E1 -23801.617,E2 -23801.617} C_VEL
LIN {X 0,Y 183.397,Z 234.762,A -85,B 0,C 180,E1 -23804.04,E2 -23804.04} C_VEL
LIN {X 0,Y 188.78,Z 247.382,A -85,B 0,C 180,E1 -23806.355,E2 -23806.355} C_VEL
LIN {X 0,Y 191.203,Z 253.812,A -85,B 0,C 180,E1 -23807.365,E2 -23807.365} C_VEL
LIN {X 0,Y 188.436,Z 299.678,A -85,B 0,C 180,E1 -23808.975,E2 -23808.975} C_VEL
LIN {X 0,Y 186.632,Z 313.347,A -85,B 0,C 180,E1 -23809.802,E2 -23809.802} C_VEL
LIN {X 0,Y 184.076,Z 326.089,A -85,B 0,C 180,E1 -23810.952,E2 -23810.952} C_VEL
LIN {X 0,Y 181.264,Z 337.152,A -85,B 0,C 180,E1 -23812.362,E2 -23812.362} C_VEL
LIN {X 0,Y 177.773,Z 348.691,A -85,B 0,C 180,E1 -23814.329,E2 -23814.329} C_VEL
LIN {X 0,Y 174.041,Z 359.081,A -85,B 0,C 180,E1 -23816.619,E2 -23816.619} C_VEL
LIN {X 0,Y 172.154,Z 363.763,A -85,B 0,C 180,E1 -23817.861,E2 -23817.861} C_VEL
LIN {X 0,Y 170.38,Z 366.654,A -85,B 0,C 180,E1 -23818.575,E2 -23818.575} C_VEL
LIN {X 0,Y 161.6,Z 375.135,A -85,B 0,C 180,E1 -23820.601,E2 -23820.601} C_VEL
LIN {X 0,Y 159.92,Z 377.564,A -85,B 0,C 180,E1 -23821.54,E2 -23821.54} C_VEL
LIN {X 0,Y 156.655,Z 384.112,A -85,B 0,C 180,E1 -23824.773,E2 -23824.773} C_VEL
LIN {X 0,Y 153.571,Z 390.051,A -85,B 0,C 180,E1 -23828.523,E2 -23828.523} C_VEL
LIN {X 0,Y 151.083,Z 394.742,A -85,B 0,C 180,E1 -23832.4,E2 -23832.4} C_VEL
LIN {X 0,Y 149.377,Z 398.325,A -85,B 0,C 180,E1 -23836.393,E2 -23836.393} C_VEL
LIN {X 0,Y 148.541,Z 400.171,A -85,B 0,C 180,E1 -23839.09,E2 -23839.09} C_VEL
LIN {X 0,Y 148.012,Z 401.555,A -85,B 0,C 180,E1 -23841.809,E2 -23841.809} C_VEL
LIN {X 0,Y 147.701,Z 402.543,A -85,B 0,C 180,E1 -23844.538,E2 -23844.538} C_VEL
LIN {X 0,Y 147.557,Z 403.145,A -85,B 0,C 180,E1 -23847.269,E2 -23847.269} C_VEL
LIN {X 0,Y 147.588,Z 403.354,A -85,B 0,C 180,E1 -23849.999,E2 -23849.999} C_VEL
LIN {X 0,Y 147.557,Z 403.13,A -85,B 0,C 180,E1 -23852.729,E2 -23852.729} C_VEL
LIN {X 0,Y 147.701,Z 402.519,A -85,B 0,C 180,E1 -23855.46,E2 -23855.46} C_VEL
LIN {X 0,Y 148.012,Z 401.521,A -85,B 0,C 180,E1 -23858.188,E2 -23858.188} C_VEL
LIN {X 0,Y 148.542,Z 400.122,A -85,B 0,C 180,E1 -23860.908,E2 -23860.908} C_VEL
LIN {X 0,Y 149.87,Z 397.188,A -85,B 0,C 180,E1 -23864.945,E2 -23864.945} C_VEL
LIN {X 0,Y 151.783,Z 393.218,A -85,B 0,C 180,E1 -23868.911,E2 -23868.911} C_VEL
LIN {X 0,Y 155.089,Z 387.115,A -85,B 0,C 180,E1 -23873.359,E2 -23873.359} C_VEL
LIN {X 0,Y 158.675,Z 380.107,A -85,B 0,C 180,E1 -23877.196,E2 -23877.196} C_VEL
LIN {X 0,Y 162.3,Z 372.176,A -85,B 0,C 180,E1 -23880.582,E2 -23880.582} C_VEL
LIN {X 0,Y 166.063,Z 363.687,A -85,B 0,C 180,E1 -23883.377,E2 -23883.377} C_VEL
LIN {X 0,Y 170.197,Z 353.197,A -85,B 0,C 180,E1 -23886.043,E2 -23886.043} C_VEL
LIN {X 0,Y 173.833,Z 342.813,A -85,B 0,C 180,E1 -23888.062,E2 -23888.062} C_VEL
LIN {X 0,Y 177.19,Z 331.416,A -85,B 0,C 180,E1 -23889.758,E2 -23889.758} C_VEL
LIN {X 0,Y 179.87,Z 319.661,A -85,B 0,C 180,E1 -23891.062,E2 -23891.062} C_VEL
LIN {X 0,Y 182.15,Z 306.677,A -85,B 0,C 180,E1 -23892.036,E2 -23892.036} C_VEL
LIN {X 0,Y 183.531,Z 292.988,A -85,B 0,C 180,E1 -23892.693,E2 -23892.693} C_VEL
LIN {X 0,Y 185.783,Z 255.858,A -85,B 0,C 180,E1 -23893.978,E2 -23893.978} C_VEL
LIN {X 0,Y 180.736,Z 242.846,A -85,B 0,C 180,E1 -23896.264,E2 -23896.264} C_VEL
LIN {X 0,Y 175.51,Z 231.746,A -85,B 0,C 180,E1 -23898.741,E2 -23898.741} C_VEL
LIN {X 0,Y 170.459,Z 222.467,A -85,B 0,C 180,E1 -23901.317,E2 -23901.317} C_VEL
LIN {X 0,Y 167.579,Z 218.009,A -85,B 0,C 180,E1 -23902.868,E2 -23902.868} C_VEL
LIN {X 0,Y 164.621,Z 213.919,A -85,B 0,C 180,E1 -23904.545,E2 -23904.545} C_VEL
LIN {X 0,Y 161.906,Z 210.105,A -85,B 0,C 180,E1 -23906.209,E2 -23906.209} C_VEL
LIN {X 0,Y 159.265,Z 206.703,A -85,B 0,C 180,E1 -23907.933,E2 -23907.933} C_VEL
LIN {X 0,Y 158.389,Z 205.481,A -85,B 0,C 180,E1 -23908.544,E2 -23908.544} C_VEL
LIN {X 0,Y 155.934,Z 202.9,A -85,B 0,C 180,E1 -23910.279,E2 -23910.279} C_VEL
LIN {X 0,Y 154.483,Z 200.435,A -85,B 0,C 180,E1 -23911.466,E2 -23911.466} C_VEL
LIN {X 0,Y 151.857,Z 198.437,A -85,B 0,C 180,E1 -23913.545,E2 -23913.545} C_VEL
LIN {X 0,Y 150.389,Z 195.641,A -85,B 0,C 180,E1 -23915.128,E2 -23915.128} C_VEL
LIN {X 0,Y 150.269,Z 194.806,A -85,B 0,C 180,E1 -23916.393,E2 -23916.393} C_VEL
LIN {X 0,Y 150.327,Z 194.739,A -85,B 0,C 180,E1 -23920.897,E2 -23920.897} C_VEL
LIN {X 0,Y 150.435,Z 194.731,A -85,B 0,C 180,E1 -23926.492,E2 -23926.492} C_VEL
LIN {X 0,Y 150.641,Z 194.694,A -85,B 0,C 180,E1 -23929.245,E2 -23929.245} C_VEL
LIN {X 0,Y 150.734,Z 194.709,A -85,B 0,C 180,E1 -23931.959,E2 -23931.959} C_VEL
LIN {X 0,Y 151.21,Z 194.636,A -85,B 0,C 180,E1 -23940,E2 -23940} C_VEL
LIN {X 0,Y 150.717,Z 194.685,A -85,B 0,C 180,E1 -23948.042,E2 -23948.042} C_VEL
LIN {X 0,Y 150.605,Z 194.71,A -85,B 0,C 180,E1 -23951.5,E2 -23951.5} C_VEL
LIN {X 0,Y 150.368,Z 194.728,A -85,B 0,C 180,E1 -23956.286,E2 -23956.286} C_VEL
LIN {X 0,Y 150.347,Z 194.738,A -85,B 0,C 180,E1 -23960.794,E2 -23960.794} C_VEL
LIN {X 0,Y 150.302,Z 195.077,A -85,B 0,C 180,E1 -23964.519,E2 -23964.519} C_VEL
LIN {X 0,Y 150.584,Z 196.242,A -85,B 0,C 180,E1 -23965.367,E2 -23965.367} C_VEL
LIN {X 0,Y 152.248,Z 198.858,A -85,B 0,C 180,E1 -23966.965,E2 -23966.965} C_VEL
LIN {X 0,Y 154.784,Z 200.711,A -85,B 0,C 180,E1 -23968.937,E2 -23968.937} C_VEL
LIN {X 0,Y 156.789,Z 204.019,A -85,B 0,C 180,E1 -23970.534,E2 -23970.534} C_VEL
LIN {X 0,Y 158.994,Z 206.105,A -85,B 0,C 180,E1 -23972.035,E2 -23972.035} C_VEL
LIN {X 0,Y 161.479,Z 209.683,A -85,B 0,C 180,E1 -23973.705,E2 -23973.705} C_VEL
LIN {X 0,Y 162.845,Z 211.361,A -85,B 0,C 180,E1 -23974.549,E2 -23974.549} C_VEL
LIN {X 0,Y 166.736,Z 216.846,A -85,B 0,C 180,E1 -23976.84,E2 -23976.84} C_VEL
LIN {X 0,Y 171.69,Z 224.012,A -85,B 0,C 180,E1 -23979.465,E2 -23979.465} C_VEL
LIN {X 0,Y 176.464,Z 231.938,A -85,B 0,C 180,E1 -23981.795,E2 -23981.795} C_VEL
LIN {X 0,Y 181.421,Z 242.479,A -85,B 0,C 180,E1 -23984.114,E2 -23984.114} C_VEL
LIN {X 0,Y 185.925,Z 253.623,A -85,B 0,C 180,E1 -23986.121,E2 -23986.121} C_VEL
LIN {X 0,Y 183.169,Z 297.074,A -85,B 0,C 180,E1 -23987.669,E2 -23987.669} C_VEL
LIN {X 0,Y 181.242,Z 310.48,A -85,B 0,C 180,E1 -23988.457,E2 -23988.457} C_VEL
LIN {X 0,Y 178.96,Z 322.671,A -85,B 0,C 180,E1 -23989.613,E2 -23989.613} C_VEL
LIN {X 0,Y 176.064,Z 333.968,A -85,B 0,C 180,E1 -23991.048,E2 -23991.048} C_VEL
LIN {X 0,Y 172.417,Z 345.606,A -85,B 0,C 180,E1 -23993.044,E2 -23993.044} C_VEL
LIN {X 0,Y 168.526,Z 356.065,A -85,B 0,C 180,E1 -23995.377,E2 -23995.377} C_VEL
LIN {X 0,Y 164.974,Z 364.611,A -85,B 0,C 180,E1 -23997.827,E2 -23997.827} C_VEL
LIN {X 0,Y 161.665,Z 372.233,A -85,B 0,C 180,E1 -24000.601,E2 -24000.601} C_VEL
LIN {X 0,Y 157.775,Z 380.182,A -85,B 0,C 180,E1 -24004.261,E2 -24004.261} C_VEL
LIN {X 0,Y 153.962,Z 387.254,A -85,B 0,C 180,E1 -24008.583,E2 -24008.583} C_VEL
LIN {X 0,Y 151.514,Z 391.962,A -85,B 0,C 180,E1 -24012.454,E2 -24012.454} C_VEL
LIN {X 0,Y 149.704,Z 395.564,A -85,B 0,C 180,E1 -24016.426,E2 -24016.426} C_VEL
LIN {X 0,Y 148.801,Z 397.424,A -85,B 0,C 180,E1 -24019.111,E2 -24019.111} C_VEL
LIN {X 0,Y 148.213,Z 398.821,A -85,B 0,C 180,E1 -24021.823,E2 -24021.823} C_VEL
LIN {X 0,Y 147.614,Z 400.425,A -85,B 0,C 180,E1 -24027.272,E2 -24027.272} C_VEL
LIN {X 0,Y 147.597,Z 400.63,A -85,B 0,C 180,E1 -24030.614,E2 -24030.614} C_VEL
LIN {X 0,Y 147.804,Z 399.866,A -85,B 0,C 180,E1 -24035.458,E2 -24035.458} C_VEL
LIN {X 0,Y 148.214,Z 398.892,A -85,B 0,C 180,E1 -24038.179,E2 -24038.179} C_VEL
LIN {X 0,Y 148.8,Z 397.526,A -85,B 0,C 180,E1 -24040.891,E2 -24040.891} C_VEL
LIN {X 0,Y 150.207,Z 394.641,A -85,B 0,C 180,E1 -24044.913,E2 -24044.913} C_VEL
LIN {X 0,Y 152.179,Z 390.73,A -85,B 0,C 180,E1 -24048.862,E2 -24048.862} C_VEL
LIN {X 0,Y 154.945,Z 385.685,A -85,B 0,C 180,E1 -24052.678,E2 -24052.678} C_VEL
LIN {X 0,Y 158.229,Z 379.334,A -85,B 0,C 180,E1 -24056.371,E2 -24056.371} C_VEL
LIN {X 0,Y 161.789,Z 371.99,A -85,B 0,C 180,E1 -24059.681,E2 -24059.681} C_VEL
LIN {X 0,Y 165.596,Z 363.295,A -85,B 0,C 180,E1 -24062.76,E2 -24062.76} C_VEL
LIN {X 0,Y 169.723,Z 353.416,A -85,B 0,C 180,E1 -24065.431,E2 -24065.431} C_VEL
LIN {X 0,Y 173.691,Z 342.29,A -85,B 0,C 180,E1 -24067.734,E2 -24067.734} C_VEL
LIN {X 0,Y 176.88,Z 331.386,A -85,B 0,C 180,E1 -24069.474,E2 -24069.474} C_VEL
LIN {X 0,Y 179.821,Z 319.33,A -85,B 0,C 180,E1 -24070.893,E2 -24070.893} C_VEL
LIN {X 0,Y 182.079,Z 306.594,A -85,B 0,C 180,E1 -24071.962,E2 -24071.962} C_VEL
LIN {X 0,Y 183.571,Z 293.717,A -85,B 0,C 180,E1 -24072.636,E2 -24072.636} C_VEL
LIN {X 0,Y 186.044,Z 253.553,A -85,B 0,C 180,E1 -24074.044,E2 -24074.044} C_VEL
LIN {X 0,Y 180.324,Z 239.664,A -85,B 0,C 180,E1 -24076.615,E2 -24076.615} C_VEL
LIN {X 0,Y 175.211,Z 229.493,A -85,B 0,C 180,E1 -24079.036,E2 -24079.036} C_VEL
LIN {X 0,Y 170.077,Z 221.625,A -85,B 0,C 180,E1 -24081.595,E2 -24081.595} C_VEL
LIN {X 0,Y 165.166,Z 214.505,A -85,B 0,C 180,E1 -24084.319,E2 -24084.319} C_VEL
LIN {X 0,Y 162.024,Z 210.167,A -85,B 0,C 180,E1 -24086.237,E2 -24086.237} C_VEL
LIN {X 0,Y 159.494,Z 207.019,A -85,B 0,C 180,E1 -24087.885,E2 -24087.885} C_VEL
LIN {X 0,Y 158.537,Z 205.531,A -85,B 0,C 180,E1 -24088.567,E2 -24088.567} C_VEL
LIN {X 0,Y 156.073,Z 203.05,A -85,B 0,C 180,E1 -24090.308,E2 -24090.308} C_VEL
LIN {X 0,Y 154.64,Z 200.497,A -85,B 0,C 180,E1 -24091.497,E2 -24091.497} C_VEL
LIN {X 0,Y 151.893,Z 198.474,A -85,B 0,C 180,E1 -24093.683,E2 -24093.683} C_VEL
LIN {X 0,Y 150.436,Z 195.787,A -85,B 0,C 180,E1 -24095.228,E2 -24095.228} C_VEL
LIN {X 0,Y 150.284,Z 194.861,A -85,B 0,C 180,E1 -24096.304,E2 -24096.304} C_VEL
LIN {X 0,Y 150.359,Z 194.755,A -85,B 0,C 180,E1 -24100.901,E2 -24100.901} C_VEL
LIN {X 0,Y 150.449,Z 194.731,A -85,B 0,C 180,E1 -24106.493,E2 -24106.493} C_VEL
LIN {X 0,Y 150.652,Z 194.697,A -85,B 0,C 180,E1 -24109.245,E2 -24109.245} C_VEL
LIN {X 0,Y 150.723,Z 194.684,A -85,B 0,C 180,E1 -24111.959,E2 -24111.959} C_VEL
LIN {X 0,Y 151.214,Z 194.635,A -85,B 0,C 180,E1 -24120,E2 -24120} C_VEL
LIN {X 0,Y 150.699,Z 194.714,A -85,B 0,C 180,E1 -24128.042,E2 -24128.042} C_VEL
LIN {X 0,Y 150.574,Z 194.701,A -85,B 0,C 180,E1 -24131.43,E2 -24131.43} C_VEL
LIN {X 0,Y 150.341,Z 194.74,A -85,B 0,C 180,E1 -24136.289,E2 -24136.289} C_VEL
LIN {X 0,Y 150.349,Z 194.756,A -85,B 0,C 180,E1 -24140.79,E2 -24140.79} C_VEL
LIN {X 0,Y 150.287,Z 194.914,A -85,B 0,C 180,E1 -24143.787,E2 -24143.787} C_VEL
LIN {X 0,Y 150.477,Z 195.907,A -85,B 0,C 180,E1 -24144.764,E2 -24144.764} C_VEL
LIN {X 0,Y 151.847,Z 198.418,A -85,B 0,C 180,E1 -24146.193,E2 -24146.193} C_VEL
LIN {X 0,Y 154.808,Z 200.793,A -85,B 0,C 180,E1 -24148.561,E2 -24148.561} C_VEL
LIN {X 0,Y 156.742,Z 203.951,A -85,B 0,C 180,E1 -24150.115,E2 -24150.115} C_VEL
LIN {X 0,Y 159.002,Z 206.17,A -85,B 0,C 180,E1 -24151.676,E2 -24151.676} C_VEL
LIN {X 0,Y 161.459,Z 209.638,A -85,B 0,C 180,E1 -24153.336,E2 -24153.336} C_VEL
LIN {X 0,Y 162.871,Z 211.348,A -85,B 0,C 180,E1 -24154.214,E2 -24154.214} C_VEL
LIN {X 0,Y 166.425,Z 216.294,A -85,B 0,C 180,E1 -24156.325,E2 -24156.325} C_VEL
LIN {X 0,Y 169.788,Z 221.26,A -85,B 0,C 180,E1 -24158.173,E2 -24158.173} C_VEL
LIN {X 0,Y 175.026,Z 230.619,A -85,B 0,C 180,E1 -24160.879,E2 -24160.879} C_VEL
LIN {X 0,Y 180.421,Z 241.934,A -85,B 0,C 180,E1 -24163.463,E2 -24163.463} C_VEL
LIN {X 0,Y 185.243,Z 254.004,A -85,B 0,C 180,E1 -24165.656,E2 -24165.656} C_VEL
LIN {X 0,Y 185.937,Z 256.385,A -85,B 0,C 180,E1 -24165.99,E2 -24165.99} C_VEL
LIN {X 0,Y 183.137,Z 299.628,A -85,B 0,C 180,E1 -24167.517,E2 -24167.517} C_VEL
LIN {X 0,Y 181.318,Z 313.043,A -85,B 0,C 180,E1 -24168.338,E2 -24168.338} C_VEL
LIN {X 0,Y 178.621,Z 326.03,A -85,B 0,C 180,E1 -24169.518,E2 -24169.518} C_VEL
LIN {X 0,Y 175.236,Z 338.674,A -85,B 0,C 180,E1 -24171.196,E2 -24171.196} C_VEL
LIN {X 0,Y 171.615,Z 349.922,A -85,B 0,C 180,E1 -24173.207,E2 -24173.207} C_VEL
LIN {X 0,Y 167.728,Z 360.05,A -85,B 0,C 180,E1 -24175.551,E2 -24175.551} C_VEL
LIN {X 0,Y 163.76,Z 369.175,A -85,B 0,C 180,E1 -24178.282,E2 -24178.282} C_VEL
LIN {X 0,Y 159.92,Z 377.564,A -85,B 0,C 180,E1 -24181.54,E2 -24181.54} C_VEL
LIN {X 0,Y 158.592,Z 379.92,A -85,B 0,C 180,E1 -24182.573,E2 -24182.573} C_VEL
LIN {X 0,Y 154.655,Z 384.31,A -85,B 0,C 180,E1 -24184.513,E2 -24184.513} C_VEL
LIN {X 0,Y 147.096,Z 390.867,A -85,B 0,C 180,E1 -24188.205,E2 -24188.205} C_VEL
LIN {X 0,Y 145.075,Z 393.254,A -85,B 0,C 180,E1 -24190.18,E2 -24190.18} C_VEL
LIN {X 0,Y 142.993,Z 397.194,A -85,B 0,C 180,E1 -24194.316,E2 -24194.316} C_VEL
LIN {X 0,Y 141.546,Z 400.106,A -85,B 0,C 180,E1 -24198.544,E2 -24198.544} C_VEL
LIN {X 0,Y 140.966,Z 401.49,A -85,B 0,C 180,E1 -24201.397,E2 -24201.397} C_VEL
LIN {X 0,Y 140.633,Z 402.479,A -85,B 0,C 180,E1 -24204.263,E2 -24204.263} C_VEL
LIN {X 0,Y 140.483,Z 403.081,A -85,B 0,C 180,E1 -24207.131,E2 -24207.131} C_VEL
LIN {X 0,Y 140.502,Z 403.289,A -85,B 0,C 180,E1 -24209.999,E2 -24209.999} C_VEL
LIN {X 0,Y 140.483,Z 403.065,A -85,B 0,C 180,E1 -24212.866,E2 -24212.866} C_VEL
LIN {X 0,Y 140.632,Z 402.454,A -85,B 0,C 180,E1 -24215.735,E2 -24215.735} C_VEL
LIN {X 0,Y 140.966,Z 401.455,A -85,B 0,C 180,E1 -24218.6,E2 -24218.6} C_VEL
LIN {X 0,Y 141.547,Z 400.056,A -85,B 0,C 180,E1 -24221.454,E2 -24221.454} C_VEL
LIN {X 0,Y 142.993,Z 397.122,A -85,B 0,C 180,E1 -24225.682,E2 -24225.682} C_VEL
LIN {X 0,Y 145.071,Z 393.152,A -85,B 0,C 180,E1 -24229.821,E2 -24229.821} C_VEL
LIN {X 0,Y 148.563,Z 387.048,A -85,B 0,C 180,E1 -24234.45,E2 -24234.45} C_VEL
LIN {X 0,Y 152.238,Z 380.316,A -85,B 0,C 180,E1 -24238.28,E2 -24238.28} C_VEL
LIN {X 0,Y 156.19,Z 372.108,A -85,B 0,C 180,E1 -24241.916,E2 -24241.916} C_VEL
LIN {X 0,Y 160.163,Z 363.619,A -85,B 0,C 180,E1 -24244.779,E2 -24244.779} C_VEL
LIN {X 0,Y 164.502,Z 353.128,A -85,B 0,C 180,E1 -24247.501,E2 -24247.501} C_VEL
LIN {X 0,Y 168.307,Z 342.744,A -85,B 0,C 180,E1 -24249.551,E2 -24249.551} C_VEL
LIN {X 0,Y 171.799,Z 331.345,A -85,B 0,C 180,E1 -24251.27,E2 -24251.27} C_VEL
LIN {X 0,Y 174.583,Z 319.588,A -85,B 0,C 180,E1 -24252.592,E2 -24252.592} C_VEL
LIN {X 0,Y 176.989,Z 306.37,A -85,B 0,C 180,E1 -24253.585,E2 -24253.585} C_VEL
LIN {X 0,Y 178.286,Z 294.03,A -85,B 0,C 180,E1 -24254.198,E2 -24254.198} C_VEL
LIN {X 0,Y 180.647,Z 258.074,A -85,B 0,C 180,E1 -24255.443,E2 -24255.443} C_VEL
LIN {X 0,Y 175.847,Z 245.658,A -85,B 0,C 180,E1 -24257.783,E2 -24257.783} C_VEL
LIN {X 0,Y 170.845,Z 234.928,A -85,B 0,C 180,E1 -24260.346,E2 -24260.346} C_VEL
LIN {X 0,Y 165.824,Z 225.638,A -85,B 0,C 180,E1 -24263.132,E2 -24263.132} C_VEL
LIN {X 0,Y 161.556,Z 219.488,A -85,B 0,C 180,E1 -24265.665,E2 -24265.665} C_VEL
LIN {X 0,Y 159.018,Z 215.903,A -85,B 0,C 180,E1 -24267.315,E2 -24267.315} C_VEL
LIN {X 0,Y 155.926,Z 211.682,A -85,B 0,C 180,E1 -24269.497,E2 -24269.497} C_VEL
LIN {X 0,Y 153.376,Z 208.752,A -85,B 0,C 180,E1 -24271.428,E2 -24271.428} C_VEL
LIN {X 0,Y 152.326,Z 206.941,A -85,B 0,C 180,E1 -24272.338,E2 -24272.338} C_VEL
LIN {X 0,Y 149.658,Z 204.614,A -85,B 0,C 180,E1 -24274.599,E2 -24274.599} C_VEL
LIN {X 0,Y 147.798,Z 201.441,A -85,B 0,C 180,E1 -24276.532,E2 -24276.532} C_VEL
LIN {X 0,Y 145.288,Z 199.75,A -85,B 0,C 180,E1 -24279.145,E2 -24279.145} C_VEL
LIN {X 0,Y 143.593,Z 197.061,A -85,B 0,C 180,E1 -24281.45,E2 -24281.45} C_VEL
LIN {X 0,Y 143.322,Z 195.912,A -85,B 0,C 180,E1 -24282.706,E2 -24282.706} C_VEL
LIN {X 0,Y 143.589,Z 195.571,A -85,B 0,C 180,E1 -24288.71,E2 -24288.71} C_VEL
LIN {X 0,Y 143.654,Z 195.587,A -85,B 0,C 180,E1 -24291.56,E2 -24291.56} C_VEL
LIN {X 0,Y 144.169,Z 195.512,A -85,B 0,C 180,E1 -24300,E2 -24300} C_VEL
LIN {X 0,Y 143.641,Z 195.564,A -85,B 0,C 180,E1 -24308.441,E2 -24308.441} C_VEL
LIN {X 0,Y 143.543,Z 195.591,A -85,B 0,C 180,E1 -24311.713,E2 -24311.713} C_VEL
LIN {X 0,Y 143.34,Z 195.873,A -85,B 0,C 180,E1 -24317.476,E2 -24317.476} C_VEL
LIN {X 0,Y 143.616,Z 196.977,A -85,B 0,C 180,E1 -24318.732,E2 -24318.732} C_VEL
LIN {X 0,Y 145.162,Z 199.601,A -85,B 0,C 180,E1 -24320.878,E2 -24320.878} C_VEL
LIN {X 0,Y 148.121,Z 201.821,A -85,B 0,C 180,E1 -24323.971,E2 -24323.971} C_VEL
LIN {X 0,Y 149.986,Z 204.99,A -85,B 0,C 180,E1 -24325.876,E2 -24325.876} C_VEL
LIN {X 0,Y 152.606,Z 207.338,A -85,B 0,C 180,E1 -24328.074,E2 -24328.074} C_VEL
LIN {X 0,Y 154.898,Z 210.721,A -85,B 0,C 180,E1 -24329.94,E2 -24329.94} C_VEL
LIN {X 0,Y 156.654,Z 212.63,A -85,B 0,C 180,E1 -24331.207,E2 -24331.207} C_VEL
LIN {X 0,Y 159.394,Z 216.309,A -85,B 0,C 180,E1 -24333.101,E2 -24333.101} C_VEL
LIN {X 0,Y 163.961,Z 222.914,A -85,B 0,C 180,E1 -24335.968,E2 -24335.968} C_VEL
LIN {X 0,Y 169.849,Z 231.845,A -85,B 0,C 180,E1 -24339.22,E2 -24339.22} C_VEL
LIN {X 0,Y 173.9,Z 239.335,A -85,B 0,C 180,E1 -24341.294,E2 -24341.294} C_VEL
LIN {X 0,Y 178.608,Z 250.231,A -85,B 0,C 180,E1 -24343.617,E2 -24343.617} C_VEL
LIN {X 0,Y 180.711,Z 255.761,A -85,B 0,C 180,E1 -24344.623,E2 -24344.623} C_VEL
LIN {X 0,Y 177.945,Z 297.48,A -85,B 0,C 180,E1 -24346.145,E2 -24346.145} C_VEL
LIN {X 0,Y 175.972,Z 310.737,A -85,B 0,C 180,E1 -24346.941,E2 -24346.941} C_VEL
LIN {X 0,Y 173.626,Z 322.743,A -85,B 0,C 180,E1 -24348.099,E2 -24348.099} C_VEL
LIN {X 0,Y 170.61,Z 334.038,A -85,B 0,C 180,E1 -24349.552,E2 -24349.552} C_VEL
LIN {X 0,Y 166.813,Z 345.675,A -85,B 0,C 180,E1 -24351.582,E2 -24351.582} C_VEL
LIN {X 0,Y 162.749,Z 356.133,A -85,B 0,C 180,E1 -24353.961,E2 -24353.961} C_VEL
LIN {X 0,Y 159,Z 364.679,A -85,B 0,C 180,E1 -24356.463,E2 -24356.463} C_VEL
LIN {X 0,Y 155.264,Z 372.821,A -85,B 0,C 180,E1 -24359.527,E2 -24359.527} C_VEL
LIN {X 0,Y 151.388,Z 380.249,A -85,B 0,C 180,E1 -24363.089,E2 -24363.089} C_VEL
LIN {X 0,Y 147.379,Z 387.321,A -85,B 0,C 180,E1 -24367.576,E2 -24367.576} C_VEL
LIN {X 0,Y 144.752,Z 392.028,A -85,B 0,C 180,E1 -24371.605,E2 -24371.605} C_VEL
LIN {X 0,Y 142.781,Z 395.63,A -85,B 0,C 180,E1 -24375.754,E2 -24375.754} C_VEL
LIN {X 0,Y 141.83,Z 397.49,A -85,B 0,C 180,E1 -24378.569,E2 -24378.569} C_VEL
LIN {X 0,Y 141.168,Z 398.887,A -85,B 0,C 180,E1 -24381.412,E2 -24381.412} C_VEL
LIN {X 0,Y 140.538,Z 400.49,A -85,B 0,C 180,E1 -24387.135,E2 -24387.135} C_VEL
LIN {X 0,Y 140.528,Z 400.718,A -85,B 0,C 180,E1 -24390.001,E2 -24390.001} C_VEL
LIN {X 0,Y 140.539,Z 400.521,A -85,B 0,C 180,E1 -24392.868,E2 -24392.868} C_VEL
LIN {X 0,Y 141.168,Z 398.956,A -85,B 0,C 180,E1 -24398.591,E2 -24398.591} C_VEL
LIN {X 0,Y 141.829,Z 397.59,A -85,B 0,C 180,E1 -24401.433,E2 -24401.433} C_VEL
LIN {X 0,Y 143.346,Z 394.705,A -85,B 0,C 180,E1 -24405.645,E2 -24405.645} C_VEL
LIN {X 0,Y 145.454,Z 390.794,A -85,B 0,C 180,E1 -24409.77,E2 -24409.77} C_VEL
LIN {X 0,Y 148.396,Z 385.749,A -85,B 0,C 180,E1 -24413.739,E2 -24413.739} C_VEL
LIN {X 0,Y 151.876,Z 379.397,A -85,B 0,C 180,E1 -24417.565,E2 -24417.565} C_VEL
LIN {X 0,Y 155.991,Z 371.307,A -85,B 0,C 180,E1 -24421.281,E2 -24421.281} C_VEL
LIN {X 0,Y 159.655,Z 363.358,A -85,B 0,C 180,E1 -24424.143,E2 -24424.143} C_VEL
LIN {X 0,Y 164.003,Z 353.477,A -85,B 0,C 180,E1 -24426.866,E2 -24426.866} C_VEL
LIN {X 0,Y 168.125,Z 342.35,A -85,B 0,C 180,E1 -24429.217,E2 -24429.217} C_VEL
LIN {X 0,Y 171.467,Z 331.445,A -85,B 0,C 180,E1 -24430.981,E2 -24430.981} C_VEL
LIN {X 0,Y 174.529,Z 319.388,A -85,B 0,C 180,E1 -24432.415,E2 -24432.415} C_VEL
LIN {X 0,Y 176.864,Z 306.749,A -85,B 0,C 180,E1 -24433.49,E2 -24433.49} C_VEL
LIN {X 0,Y 178.459,Z 293.291,A -85,B 0,C 180,E1 -24434.197,E2 -24434.197} C_VEL
LIN {X 0,Y 180.876,Z 255.765,A -85,B 0,C 180,E1 -24435.528,E2 -24435.528} C_VEL
LIN {X 0,Y 175.796,Z 243.293,A -85,B 0,C 180,E1 -24437.985,E2 -24437.985} C_VEL
LIN {X 0,Y 171.219,Z 234.056,A -85,B 0,C 180,E1 -24440.308,E2 -24440.308} C_VEL
LIN {X 0,Y 165.128,Z 224.419,A -85,B 0,C 180,E1 -24443.618,E2 -24443.618} C_VEL
LIN {X 0,Y 159.251,Z 216.105,A -85,B 0,C 180,E1 -24447.274,E2 -24447.274} C_VEL
LIN {X 0,Y 156.446,Z 212.249,A -85,B 0,C 180,E1 -24449.249,E2 -24449.249} C_VEL
LIN {X 0,Y 153.254,Z 208.496,A -85,B 0,C 180,E1 -24451.683,E2 -24451.683} C_VEL
LIN {X 0,Y 152.299,Z 206.899,A -85,B 0,C 180,E1 -24452.518,E2 -24452.518} C_VEL
LIN {X 0,Y 149.591,Z 204.492,A -85,B 0,C 180,E1 -24454.853,E2 -24454.853} C_VEL
LIN {X 0,Y 147.986,Z 201.557,A -85,B 0,C 180,E1 -24456.563,E2 -24456.563} C_VEL
LIN {X 0,Y 145.16,Z 199.595,A -85,B 0,C 180,E1 -24459.565,E2 -24459.565} C_VEL
LIN {X 0,Y 143.473,Z 196.602,A -85,B 0,C 180,E1 -24462.08,E2 -24462.08} C_VEL
LIN {X 0,Y 143.325,Z 195.699,A -85,B 0,C 180,E1 -24463.623,E2 -24463.623} C_VEL
LIN {X 0,Y 143.595,Z 195.58,A -85,B 0,C 180,E1 -24468.71,E2 -24468.71} C_VEL
LIN {X 0,Y 143.647,Z 195.563,A -85,B 0,C 180,E1 -24471.56,E2 -24471.56} C_VEL
LIN {X 0,Y 144.173,Z 195.511,A -85,B 0,C 180,E1 -24480,E2 -24480} C_VEL
LIN {X 0,Y 143.621,Z 195.591,A -85,B 0,C 180,E1 -24488.442,E2 -24488.442} C_VEL
LIN {X 0,Y 143.5,Z 195.582,A -85,B 0,C 180,E1 -24491.619,E2 -24491.619} C_VEL
LIN {X 0,Y 143.305,Z 195.868,A -85,B 0,C 180,E1 -24496.746,E2 -24496.746} C_VEL
LIN {X 0,Y 143.563,Z 196.962,A -85,B 0,C 180,E1 -24498.092,E2 -24498.092} C_VEL
LIN {X 0,Y 145.219,Z 199.675,A -85,B 0,C 180,E1 -24500.426,E2 -24500.426} C_VEL
LIN {X 0,Y 148.124,Z 201.812,A -85,B 0,C 180,E1 -24503.506,E2 -24503.506} C_VEL
LIN {X 0,Y 149.781,Z 204.748,A -85,B 0,C 180,E1 -24505.245,E2 -24505.245} C_VEL
LIN {X 0,Y 152.641,Z 207.392,A -85,B 0,C 180,E1 -24507.693,E2 -24507.693} C_VEL
LIN {X 0,Y 155.012,Z 210.849,A -85,B 0,C 180,E1 -24509.635,E2 -24509.635} C_VEL
LIN {X 0,Y 156.603,Z 212.565,A -85,B 0,C 180,E1 -24510.792,E2 -24510.792} C_VEL
LIN {X 0,Y 159.347,Z 216.185,A -85,B 0,C 180,E1 -24512.703,E2 -24512.703} C_VEL
LIN {X 0,Y 164.08,Z 223.016,A -85,B 0,C 180,E1 -24515.695,E2 -24515.695} C_VEL
LIN {X 0,Y 167.162,Z 227.773,A -85,B 0,C 180,E1 -24517.468,E2 -24517.468} C_VEL
LIN {X 0,Y 172.651,Z 238.378,A -85,B 0,C 180,E1 -24520.451,E2 -24520.451} C_VEL
LIN {X 0,Y 177.278,Z 248.846,A -85,B 0,C 180,E1 -24522.787,E2 -24522.787} C_VEL
LIN {X 0,Y 180.744,Z 258.063,A -85,B 0,C 180,E1 -24524.473,E2 -24524.473} C_VEL
LIN {X 0,Y 177.93,Z 299.871,A -85,B 0,C 180,E1 -24525.987,E2 -24525.987} C_VEL
LIN {X 0,Y 176.046,Z 313.227,A -85,B 0,C 180,E1 -24526.823,E2 -24526.823} C_VEL
LIN {X 0,Y 173.286,Z 325.972,A -85,B 0,C 180,E1 -24527.995,E2 -24527.995} C_VEL
LIN {X 0,Y 170.231,Z 337.032,A -85,B 0,C 180,E1 -24529.44,E2 -24529.44} C_VEL
LIN {X 0,Y 166.442,Z 348.569,A -85,B 0,C 180,E1 -24531.478,E2 -24531.478} C_VEL
LIN {X 0,Y 162.355,Z 358.958,A -85,B 0,C 180,E1 -24533.857,E2 -24533.857} C_VEL
LIN {X 0,Y 158.538,Z 367.449,A -85,B 0,C 180,E1 -24536.349,E2 -24536.349} C_VEL
LIN {X 0,Y 154.807,Z 375.283,A -85,B 0,C 180,E1 -24539.287,E2 -24539.287} C_VEL
LIN {X 0,Y 150.907,Z 382.932,A -85,B 0,C 180,E1 -24542.994,E2 -24542.994} C_VEL
LIN {X 0,Y 146.978,Z 389.988,A -85,B 0,C 180,E1 -24547.509,E2 -24547.509} C_VEL
LIN {X 0,Y 145.075,Z 393.254,A -85,B 0,C 180,E1 -24550.18,E2 -24550.18} C_VEL
LIN {X 0,Y 143.255,Z 395.44,A -85,B 0,C 180,E1 -24552.249,E2 -24552.249} C_VEL
LIN {X 0,Y 138.879,Z 398.447,A -85,B 0,C 180,E1 -24555.65,E2 -24555.65} C_VEL
LIN {X 0,Y 135.551,Z 400.329,A -85,B 0,C 180,E1 -24558.562,E2 -24558.562} C_VEL
LIN {X 0,Y 134.002,Z 401.427,A -85,B 0,C 180,E1 -24560.948,E2 -24560.948} C_VEL
LIN {X 0,Y 133.786,Z 401.7,A -85,B 0,C 180,E1 -24561.778,E2 -24561.778} C_VEL
LIN {X 0,Y 133.399,Z 403.016,A -85,B 0,C 180,E1 -24566.979,E2 -24566.979} C_VEL
LIN {X 0,Y 133.418,Z 403.224,A -85,B 0,C 180,E1 -24569.999,E2 -24569.999} C_VEL
LIN {X 0,Y 133.398,Z 403,A -85,B 0,C 180,E1 -24573.019,E2 -24573.019} C_VEL
LIN {X 0,Y 133.56,Z 402.388,A -85,B 0,C 180,E1 -24576.04,E2 -24576.04} C_VEL
LIN {X 0,Y 133.924,Z 401.39,A -85,B 0,C 180,E1 -24579.056,E2 -24579.056} C_VEL
LIN {X 0,Y 134.573,Z 399.99,A -85,B 0,C 180,E1 -24582.056,E2 -24582.056} C_VEL
LIN {X 0,Y 136.146,Z 397.056,A -85,B 0,C 180,E1 -24586.492,E2 -24586.492} C_VEL
LIN {X 0,Y 138.404,Z 393.086,A -85,B 0,C 180,E1 -24590.819,E2 -24590.819} C_VEL
LIN {X 0,Y 142.097,Z 386.982,A -85,B 0,C 180,E1 -24595.641,E2 -24595.641} C_VEL
LIN {X 0,Y 146.375,Z 379.507,A -85,B 0,C 180,E1 -24599.998,E2 -24599.998} C_VEL
LIN {X 0,Y 150.192,Z 372.041,A -85,B 0,C 180,E1 -24603.353,E2 -24603.353} C_VEL
LIN {X 0,Y 154.378,Z 363.551,A -85,B 0,C 180,E1 -24606.284,E2 -24606.284} C_VEL
LIN {X 0,Y 158.929,Z 353.06,A -85,B 0,C 180,E1 -24609.058,E2 -24609.058} C_VEL
LIN {X 0,Y 162.902,Z 342.675,A -85,B 0,C 180,E1 -24611.139,E2 -24611.139} C_VEL
LIN {X 0,Y 166.538,Z 331.275,A -85,B 0,C 180,E1 -24612.879,E2 -24612.879} C_VEL
LIN {X 0,Y 169.431,Z 319.515,A -85,B 0,C 180,E1 -24614.214,E2 -24614.214} C_VEL
LIN {X 0,Y 171.929,Z 306.236,A -85,B 0,C 180,E1 -24615.219,E2 -24615.219} C_VEL
LIN {X 0,Y 173.318,Z 293.519,A -85,B 0,C 180,E1 -24615.847,E2 -24615.847} C_VEL
LIN {X 0,Y 175.525,Z 260.161,A -85,B 0,C 180,E1 -24617.04,E2 -24617.04} C_VEL
LIN {X 0,Y 171.343,Z 249.065,A -85,B 0,C 180,E1 -24619.251,E2 -24619.251} C_VEL
LIN {X 0,Y 167.025,Z 239.531,A -85,B 0,C 180,E1 -24621.637,E2 -24621.637} C_VEL
LIN {X 0,Y 162.227,Z 230.413,A -85,B 0,C 180,E1 -24624.498,E2 -24624.498} C_VEL
LIN {X 0,Y 156.484,Z 222.011,A -85,B 0,C 180,E1 -24628.261,E2 -24628.261} C_VEL
LIN {X 0,Y 153.194,Z 217.582,A -85,B 0,C 180,E1 -24630.714,E2 -24630.714} C_VEL
LIN {X 0,Y 150.544,Z 214.037,A -85,B 0,C 180,E1 -24632.921,E2 -24632.921} C_VEL
LIN {X 0,Y 149.819,Z 213.143,A -85,B 0,C 180,E1 -24633.56,E2 -24633.56} C_VEL
LIN {X 0,Y 147.085,Z 210.143,A -85,B 0,C 180,E1 -24636.131,E2 -24636.131} C_VEL
LIN {X 0,Y 146.006,Z 208.135,A -85,B 0,C 180,E1 -24637.351,E2 -24637.351} C_VEL
LIN {X 0,Y 143.511,Z 206.188,A -85,B 0,C 180,E1 -24640.139,E2 -24640.139} C_VEL
LIN {X 0,Y 141.751,Z 203.178,A -85,B 0,C 180,E1 -24642.694,E2 -24642.694} C_VEL
LIN {X 0,Y 140.842,Z 202.318,A -85,B 0,C 180,E1 -24644.071,E2 -24644.071} C_VEL
LIN {X 0,Y 138.33,Z 200.341,A -85,B 0,C 180,E1 -24648.724,E2 -24648.724} C_VEL
LIN {X 0,Y 136.741,Z 197.247,A -85,B 0,C 180,E1 -24654.84,E2 -24654.84} C_VEL
LIN {X 0,Y 137.126,Z 196.458,A -85,B 0,C 180,E1 -24660,E2 -24660} C_VEL
LIN {X 0,Y 136.753,Z 197.388,A -85,B 0,C 180,E1 -24665.715,E2 -24665.715} C_VEL
LIN {X 0,Y 139.672,Z 201.66,A -85,B 0,C 180,E1 -24674.2,E2 -24674.2} C_VEL
LIN {X 0,Y 141.719,Z 202.967,A -85,B 0,C 180,E1 -24677.403,E2 -24677.403} C_VEL
LIN {X 0,Y 143.261,Z 205.868,A -85,B 0,C 180,E1 -24679.711,E2 -24679.711} C_VEL
LIN {X 0,Y 145.856,Z 208.078,A -85,B 0,C 180,E1 -24682.674,E2 -24682.674} C_VEL
LIN {X 0,Y 146.584,Z 209.228,A -85,B 0,C 180,E1 -24683.488,E2 -24683.488} C_VEL
LIN {X 0,Y 149.025,Z 212.443,A -85,B 0,C 180,E1 -24685.92,E2 -24685.92} C_VEL
LIN {X 0,Y 150.467,Z 213.839,A -85,B 0,C 180,E1 -24687.176,E2 -24687.176} C_VEL
LIN {X 0,Y 153.045,Z 217.425,A -85,B 0,C 180,E1 -24689.345,E2 -24689.345} C_VEL
LIN {X 0,Y 154.348,Z 219.07,A -85,B 0,C 180,E1 -24690.346,E2 -24690.346} C_VEL
LIN {X 0,Y 157.842,Z 224.03,A -85,B 0,C 180,E1 -24692.865,E2 -24692.865} C_VEL
LIN {X 0,Y 162.241,Z 230.409,A -85,B 0,C 180,E1 -24695.682,E2 -24695.682} C_VEL
LIN {X 0,Y 167.982,Z 239.916,A -85,B 0,C 180,E1 -24698.972,E2 -24698.972} C_VEL
LIN {X 0,Y 172.188,Z 249,A -85,B 0,C 180,E1 -24701.243,E2 -24701.243} C_VEL
LIN {X 0,Y 175.682,Z 258.04,A -85,B 0,C 180,E1 -24703.064,E2 -24703.064} C_VEL
LIN {X 0,Y 172.98,Z 297.071,A -85,B 0,C 180,E1 -24704.499,E2 -24704.499} C_VEL
LIN {X 0,Y 170.983,Z 310.268,A -85,B 0,C 180,E1 -24705.285,E2 -24705.285} C_VEL
LIN {X 0,Y 168.423,Z 322.815,A -85,B 0,C 180,E1 -24706.49,E2 -24706.49} C_VEL
LIN {X 0,Y 165.282,Z 334.108,A -85,B 0,C 180,E1 -24707.958,E2 -24707.958} C_VEL
LIN {X 0,Y 161.32,Z 345.744,A -85,B 0,C 180,E1 -24710.017,E2 -24710.017} C_VEL
LIN {X 0,Y 157.075,Z 356.201,A -85,B 0,C 180,E1 -24712.44,E2 -24712.44} C_VEL
LIN {X 0,Y 153.126,Z 364.747,A -85,B 0,C 180,E1 -24714.993,E2 -24714.993} C_VEL
LIN {X 0,Y 148.908,Z 373.401,A -85,B 0,C 180,E1 -24718.371,E2 -24718.371} C_VEL
LIN {X 0,Y 144.46,Z 381.429,A -85,B 0,C 180,E1 -24722.474,E2 -24722.474} C_VEL
LIN {X 0,Y 140.848,Z 387.387,A -85,B 0,C 180,E1 -24726.475,E2 -24726.475} C_VEL
LIN {X 0,Y 138.001,Z 392.095,A -85,B 0,C 180,E1 -24730.671,E2 -24730.671} C_VEL
LIN {X 0,Y 135.893,Z 395.696,A -85,B 0,C 180,E1 -24735.016,E2 -24735.016} C_VEL
LIN {X 0,Y 134.857,Z 397.556,A -85,B 0,C 180,E1 -24737.97,E2 -24737.97} C_VEL
LIN {X 0,Y 134.138,Z 398.952,A -85,B 0,C 180,E1 -24740.958,E2 -24740.958} C_VEL
LIN {X 0,Y 133.466,Z 400.555,A -85,B 0,C 180,E1 -24746.983,E2 -24746.983} C_VEL
LIN {X 0,Y 133.45,Z 400.783,A -85,B 0,C 180,E1 -24750.001,E2 -24750.001} C_VEL
LIN {X 0,Y 133.466,Z 400.586,A -85,B 0,C 180,E1 -24753.02,E2 -24753.02} C_VEL
LIN {X 0,Y 134.138,Z 399.021,A -85,B 0,C 180,E1 -24759.044,E2 -24759.044} C_VEL
LIN {X 0,Y 134.857,Z 397.655,A -85,B 0,C 180,E1 -24762.033,E2 -24762.033} C_VEL
LIN {X 0,Y 136.519,Z 394.769,A -85,B 0,C 180,E1 -24766.449,E2 -24766.449} C_VEL
LIN {X 0,Y 138.768,Z 390.858,A -85,B 0,C 180,E1 -24770.765,E2 -24770.765} C_VEL
LIN {X 0,Y 141.911,Z 385.813,A -85,B 0,C 180,E1 -24774.895,E2 -24774.895} C_VEL
LIN {X 0,Y 145.605,Z 379.46,A -85,B 0,C 180,E1 -24778.861,E2 -24778.861} C_VEL
LIN {X 0,Y 149.88,Z 371.519,A -85,B 0,C 180,E1 -24782.631,E2 -24782.631} C_VEL
LIN {X 0,Y 153.822,Z 363.42,A -85,B 0,C 180,E1 -24785.629,E2 -24785.629} C_VEL
LIN {X 0,Y 158.383,Z 353.538,A -85,B 0,C 180,E1 -24788.406,E2 -24788.406} C_VEL
LIN {X 0,Y 162.699,Z 342.411,A -85,B 0,C 180,E1 -24790.794,E2 -24790.794} C_VEL
LIN {X 0,Y 166.181,Z 331.504,A -85,B 0,C 180,E1 -24792.583,E2 -24792.583} C_VEL
LIN {X 0,Y 169.371,Z 319.445,A -85,B 0,C 180,E1 -24794.03,E2 -24794.03} C_VEL
LIN {X 0,Y 171.846,Z 306.486,A -85,B 0,C 180,E1 -24795.134,E2 -24795.134} C_VEL
LIN {X 0,Y 173.463,Z 293.074,A -85,B 0,C 180,E1 -24795.842,E2 -24795.842} C_VEL
LIN {X 0,Y 175.82,Z 258.039,A -85,B 0,C 180,E1 -24797.101,E2 -24797.101} C_VEL
LIN {X 0,Y 171.208,Z 246.515,A -85,B 0,C 180,E1 -24799.516,E2 -24799.516} C_VEL
LIN {X 0,Y 167.346,Z 238.647,A -85,B 0,C 180,E1 -24801.624,E2 -24801.624} C_VEL
LIN {X 0,Y 162.993,Z 231.632,A -85,B 0,C 180,E1 -24804.116,E2 -24804.116} C_VEL
LIN {X 0,Y 158.677,Z 225.145,A -85,B 0,C 180,E1 -24806.856,E2 -24806.856} C_VEL
LIN {X 0,Y 156.161,Z 221.543,A -85,B 0,C 180,E1 -24808.611,E2 -24808.611} C_VEL
LIN {X 0,Y 153.371,Z 217.724,A -85,B 0,C 180,E1 -24810.723,E2 -24810.723} C_VEL
LIN {X 0,Y 150.58,Z 213.971,A -85,B 0,C 180,E1 -24813.066,E2 -24813.066} C_VEL
LIN {X 0,Y 149.353,Z 212.74,A -85,B 0,C 180,E1 -24814.142,E2 -24814.142} C_VEL
LIN {X 0,Y 146.891,Z 209.729,A -85,B 0,C 180,E1 -24816.565,E2 -24816.565} C_VEL
LIN {X 0,Y 146.049,Z 208.153,A -85,B 0,C 180,E1 -24817.539,E2 -24817.539} C_VEL
LIN {X 0,Y 143.326,Z 205.938,A -85,B 0,C 180,E1 -24820.671,E2 -24820.671} C_VEL
LIN {X 0,Y 141.43,Z 202.59,A -85,B 0,C 180,E1 -24823.583,E2 -24823.583} C_VEL
LIN {X 0,Y 138.274,Z 200.299,A -85,B 0,C 180,E1 -24829.495,E2 -24829.495} C_VEL
LIN {X 0,Y 136.831,Z 197.244,A -85,B 0,C 180,E1 -24836.319,E2 -24836.319} C_VEL
LIN {X 0,Y 137.135,Z 196.581,A -85,B 0,C 180,E1 -24840,E2 -24840} C_VEL
LIN {X 0,Y 136.824,Z 197.499,A -85,B 0,C 180,E1 -24844.419,E2 -24844.419} C_VEL
LIN {X 0,Y 140.26,Z 202.035,A -85,B 0,C 180,E1 -24854.509,E2 -24854.509} C_VEL
LIN {X 0,Y 141.693,Z 202.972,A -85,B 0,C 180,E1 -24856.756,E2 -24856.756} C_VEL
LIN {X 0,Y 143.387,Z 205.977,A -85,B 0,C 180,E1 -24859.32,E2 -24859.32} C_VEL
LIN {X 0,Y 146.012,Z 208.165,A -85,B 0,C 180,E1 -24862.344,E2 -24862.344} C_VEL
LIN {X 0,Y 148.359,Z 211.781,A -85,B 0,C 180,E1 -24864.861,E2 -24864.861} C_VEL
LIN {X 0,Y 150.498,Z 213.887,A -85,B 0,C 180,E1 -24866.78,E2 -24866.78} C_VEL
LIN {X 0,Y 153.309,Z 217.693,A -85,B 0,C 180,E1 -24869.148,E2 -24869.148} C_VEL
LIN {X 0,Y 157.537,Z 223.448,A -85,B 0,C 180,E1 -24872.277,E2 -24872.277} C_VEL
LIN {X 0,Y 162.544,Z 230.838,A -85,B 0,C 180,E1 -24875.521,E2 -24875.521} C_VEL
LIN {X 0,Y 167.425,Z 240.13,A -85,B 0,C 180,E1 -24878.427,E2 -24878.427} C_VEL
LIN {X 0,Y 172.324,Z 251.124,A -85,B 0,C 180,E1 -24881.12,E2 -24881.12} C_VEL
LIN {X 0,Y 175.698,Z 260.255,A -85,B 0,C 180,E1 -24882.903,E2 -24882.903} C_VEL
LIN {X 0,Y 172.969,Z 299.332,A -85,B 0,C 180,E1 -24884.333,E2 -24884.333} C_VEL
LIN {X 0,Y 171.043,Z 312.627,A -85,B 0,C 180,E1 -24885.156,E2 -24885.156} C_VEL
LIN {X 0,Y 168.368,Z 324.813,A -85,B 0,C 180,E1 -24886.263,E2 -24886.263} C_VEL
LIN {X 0,Y 164.914,Z 336.972,A -85,B 0,C 180,E1 -24887.84,E2 -24887.84} C_VEL
LIN {X 0,Y 160.952,Z 348.508,A -85,B 0,C 180,E1 -24889.904,E2 -24889.904} C_VEL
LIN {X 0,Y 156.655,Z 358.896,A -85,B 0,C 180,E1 -24892.319,E2 -24892.319} C_VEL
LIN {X 0,Y 152.672,Z 367.387,A -85,B 0,C 180,E1 -24894.871,E2 -24894.871} C_VEL
LIN {X 0,Y 148.712,Z 375.22,A -85,B 0,C 180,E1 -24897.881,E2 -24897.881} C_VEL
LIN {X 0,Y 144.62,Z 382.869,A -85,B 0,C 180,E1 -24901.717,E2 -24901.717} C_VEL
LIN {X 0,Y 141.566,Z 388.111,A -85,B 0,C 180,E1 -24905.04,E2 -24905.04} C_VEL
LIN {X 0,Y 138.236,Z 393.468,A -85,B 0,C 180,E1 -24909.459,E2 -24909.459} C_VEL
LIN {X 0,Y 135.545,Z 398.196,A -85,B 0,C 180,E1 -24914.973,E2 -24914.973} C_VEL
LIN {X 0,Y 134.572,Z 400.042,A -85,B 0,C 180,E1 -24917.941,E2 -24917.941} C_VEL
LIN {X 0,Y 133.786,Z 401.7,A -85,B 0,C 180,E1 -24921.778,E2 -24921.778} C_VEL
LIN {X 0,Y 132.817,Z 402.511,A -85,B 0,C 180,E1 -24924.264,E2 -24924.264} C_VEL
LIN {X 0,Y 131.057,Z 402.977,A -85,B 0,C 180,E1 -24926.726,E2 -24926.726} C_VEL
LIN {X 0,Y 127.307,Z 403.081,A -85,B 0,C 180,E1 -24931.792,E2 -24931.792} C_VEL
LIN {X 0,Y 126.4,Z 402.742,A -85,B 0,C 180,E1 -24934.465,E2 -24934.465} C_VEL
LIN {X 0,Y 126.384,Z 402.517,A -85,B 0,C 180,E1 -24935.368,E2 -24935.368} C_VEL
LIN {X 0,Y 126.907,Z 401.324,A -85,B 0,C 180,E1 -24939.562,E2 -24939.562} C_VEL
LIN {X 0,Y 127.625,Z 399.924,A -85,B 0,C 180,E1 -24942.723,E2 -24942.723} C_VEL
LIN {X 0,Y 129.334,Z 396.99,A -85,B 0,C 180,E1 -24947.388,E2 -24947.388} C_VEL
LIN {X 0,Y 131.789,Z 393.02,A -85,B 0,C 180,E1 -24951.917,E2 -24951.917} C_VEL
LIN {X 0,Y 135.684,Z 386.915,A -85,B 0,C 180,E1 -24956.948,E2 -24956.948} C_VEL
LIN {X 0,Y 139.919,Z 379.999,A -85,B 0,C 180,E1 -24961.154,E2 -24961.154} C_VEL
LIN {X 0,Y 144.295,Z 371.973,A -85,B 0,C 180,E1 -24964.908,E2 -24964.908} C_VEL
LIN {X 0,Y 148.714,Z 363.483,A -85,B 0,C 180,E1 -24967.903,E2 -24967.903} C_VEL
LIN {X 0,Y 153.487,Z 352.991,A -85,B 0,C 180,E1 -24970.727,E2 -24970.727} C_VEL
LIN {X 0,Y 157.634,Z 342.606,A -85,B 0,C 180,E1 -24972.834,E2 -24972.834} C_VEL
LIN {X 0,Y 161.404,Z 331.204,A -85,B 0,C 180,E1 -24974.595,E2 -24974.595} C_VEL
LIN {X 0,Y 164.424,Z 319.442,A -85,B 0,C 180,E1 -24975.938,E2 -24975.938} C_VEL
LIN {X 0,Y 167.029,Z 306.072,A -85,B 0,C 180,E1 -24976.95,E2 -24976.95} C_VEL
LIN {X 0,Y 168.518,Z 292.388,A -85,B 0,C 180,E1 -24977.623,E2 -24977.623} C_VEL
LIN {X 0,Y 170.615,Z 262.334,A -85,B 0,C 180,E1 -24978.7,E2 -24978.7} C_VEL
LIN {X 0,Y 167.018,Z 252.61,A -85,B 0,C 180,E1 -24980.762,E2 -24980.762} C_VEL
LIN {X 0,Y 162.78,Z 243.133,A -85,B 0,C 180,E1 -24983.299,E2 -24983.299} C_VEL
LIN {X 0,Y 158.919,Z 235.616,A -85,B 0,C 180,E1 -24985.789,E2 -24985.789} C_VEL
LIN {X 0,Y 153.833,Z 227.914,A -85,B 0,C 180,E1 -24989.357,E2 -24989.357} C_VEL
LIN {X 0,Y 150.726,Z 223.628,A -85,B 0,C 180,E1 -24991.825,E2 -24991.825} C_VEL
LIN {X 0,Y 147.779,Z 219.577,A -85,B 0,C 180,E1 -24994.473,E2 -24994.473} C_VEL
LIN {X 0,Y 144.956,Z 216.184,A -85,B 0,C 180,E1 -24997.331,E2 -24997.331} C_VEL
LIN {X 0,Y 144.285,Z 214.835,A -85,B 0,C 180,E1 -24998.15,E2 -24998.15} C_VEL
LIN {X 0,Y 141.627,Z 212.406,A -85,B 0,C 180,E1 -25001.37,E2 -25001.37} C_VEL
LIN {X 0,Y 140.004,Z 209.42,A -85,B 0,C 180,E1 -25003.973,E2 -25003.973} C_VEL
LIN {X 0,Y 137.333,Z 207.411,A -85,B 0,C 180,E1 -25008.958,E2 -25008.958} C_VEL
LIN {X 0,Y 135.526,Z 204.02,A -85,B 0,C 180,E1 -25015.911,E2 -25015.911} C_VEL
LIN {X 0,Y 135.253,Z 203.318,A -85,B 0,C 180,E1 -25020,E2 -25020} C_VEL
LIN {X 0,Y 135.731,Z 204.487,A -85,B 0,C 180,E1 -25025.572,E2 -25025.572} C_VEL
LIN {X 0,Y 138.726,Z 208.711,A -85,B 0,C 180,E1 -25034.112,E2 -25034.112} C_VEL
LIN {X 0,Y 140.202,Z 209.647,A -85,B 0,C 180,E1 -25036.518,E2 -25036.518} C_VEL
LIN {X 0,Y 141.853,Z 212.691,A -85,B 0,C 180,E1 -25039.115,E2 -25039.115} C_VEL
LIN {X 0,Y 144.476,Z 215.253,A -85,B 0,C 180,E1 -25042.264,E2 -25042.264} C_VEL
LIN {X 0,Y 147.01,Z 218.866,A -85,B 0,C 180,E1 -25044.987,E2 -25044.987} C_VEL
LIN {X 0,Y 148.427,Z 220.376,A -85,B 0,C 180,E1 -25046.304,E2 -25046.304} C_VEL
LIN {X 0,Y 151.252,Z 224.146,A -85,B 0,C 180,E1 -25048.767,E2 -25048.767} C_VEL
LIN {X 0,Y 155.484,Z 230.434,A -85,B 0,C 180,E1 -25052.042,E2 -25052.042} C_VEL
LIN {X 0,Y 159.594,Z 236.767,A -85,B 0,C 180,E1 -25054.827,E2 -25054.827} C_VEL
LIN {X 0,Y 164.484,Z 245.083,A -85,B 0,C 180,E1 -25057.798,E2 -25057.798} C_VEL
LIN {X 0,Y 168.545,Z 254.404,A -85,B 0,C 180,E1 -25060.157,E2 -25060.157} C_VEL
LIN {X 0,Y 170.748,Z 260.149,A -85,B 0,C 180,E1 -25061.388,E2 -25061.388} C_VEL
LIN {X 0,Y 168.095,Z 297.099,A -85,B 0,C 180,E1 -25062.773,E2 -25062.773} C_VEL
LIN {X 0,Y 165.97,Z 310.595,A -85,B 0,C 180,E1 -25063.581,E2 -25063.581} C_VEL
LIN {X 0,Y 163.358,Z 322.887,A -85,B 0,C 180,E1 -25064.779,E2 -25064.779} C_VEL
LIN {X 0,Y 160.093,Z 334.178,A -85,B 0,C 180,E1 -25066.26,E2 -25066.26} C_VEL
LIN {X 0,Y 155.96,Z 345.813,A -85,B 0,C 180,E1 -25068.345,E2 -25068.345} C_VEL
LIN {X 0,Y 151.506,Z 356.27,A -85,B 0,C 180,E1 -25070.803,E2 -25070.803} C_VEL
LIN {X 0,Y 147.354,Z 364.815,A -85,B 0,C 180,E1 -25073.406,E2 -25073.406} C_VEL
LIN {X 0,Y 143.446,Z 372.414,A -85,B 0,C 180,E1 -25076.398,E2 -25076.398} C_VEL
LIN {X 0,Y 138.824,Z 380.383,A -85,B 0,C 180,E1 -25080.425,E2 -25080.425} C_VEL
LIN {X 0,Y 134.372,Z 387.453,A -85,B 0,C 180,E1 -25085.267,E2 -25085.267} C_VEL
LIN {X 0,Y 131.299,Z 392.161,A -85,B 0,C 180,E1 -25089.642,E2 -25089.642} C_VEL
LIN {X 0,Y 129.041,Z 395.762,A -85,B 0,C 180,E1 -25094.2,E2 -25094.2} C_VEL
LIN {X 0,Y 127.913,Z 397.621,A -85,B 0,C 180,E1 -25097.306,E2 -25097.306} C_VEL
LIN {X 0,Y 127.131,Z 399.017,A -85,B 0,C 180,E1 -25100.455,E2 -25100.455} C_VEL
LIN {X 0,Y 126.382,Z 400.62,A -85,B 0,C 180,E1 -25106.814,E2 -25106.814} C_VEL
LIN {X 0,Y 126.362,Z 400.848,A -85,B 0,C 180,E1 -25110.001,E2 -25110.001} C_VEL
LIN {X 0,Y 126.383,Z 400.65,A -85,B 0,C 180,E1 -25113.189,E2 -25113.189} C_VEL
LIN {X 0,Y 127.132,Z 399.085,A -85,B 0,C 180,E1 -25119.547,E2 -25119.547} C_VEL
LIN {X 0,Y 127.912,Z 397.719,A -85,B 0,C 180,E1 -25122.697,E2 -25122.697} C_VEL
LIN {X 0,Y 129.706,Z 394.833,A -85,B 0,C 180,E1 -25127.339,E2 -25127.339} C_VEL
LIN {X 0,Y 132.129,Z 390.922,A -85,B 0,C 180,E1 -25131.86,E2 -25131.86} C_VEL
LIN {X 0,Y 135.495,Z 385.876,A -85,B 0,C 180,E1 -25136.161,E2 -25136.161} C_VEL
LIN {X 0,Y 139.424,Z 379.523,A -85,B 0,C 180,E1 -25140.271,E2 -25140.271} C_VEL
LIN {X 0,Y 143.77,Z 371.876,A -85,B 0,C 180,E1 -25144.037,E2 -25144.037} C_VEL
LIN {X 0,Y 148.114,Z 363.482,A -85,B 0,C 180,E1 -25147.228,E2 -25147.228} C_VEL
LIN {X 0,Y 152.885,Z 353.6,A -85,B 0,C 180,E1 -25150.059,E2 -25150.059} C_VEL
LIN {X 0,Y 157.402,Z 342.471,A -85,B 0,C 180,E1 -25152.48,E2 -25152.48} C_VEL
LIN {X 0,Y 161.031,Z 331.563,A -85,B 0,C 180,E1 -25154.291,E2 -25154.291} C_VEL
LIN {X 0,Y 164.355,Z 319.502,A -85,B 0,C 180,E1 -25155.746,E2 -25155.746} C_VEL
LIN {X 0,Y 166.806,Z 307.279,A -85,B 0,C 180,E1 -25156.811,E2 -25156.811} C_VEL
LIN {X 0,Y 168.52,Z 294.193,A -85,B 0,C 180,E1 -25157.522,E2 -25157.522} C_VEL
LIN {X 0,Y 170.903,Z 260.305,A -85,B 0,C 180,E1 -25158.767,E2 -25158.767} C_VEL
LIN {X 0,Y 166.811,Z 249.907,A -85,B 0,C 180,E1 -25161.094,E2 -25161.094} C_VEL
LIN {X 0,Y 163.618,Z 243.354,A -85,B 0,C 180,E1 -25162.968,E2 -25162.968} C_VEL
LIN {X 0,Y 158.62,Z 235.084,A -85,B 0,C 180,E1 -25166.089,E2 -25166.089} C_VEL
LIN {X 0,Y 154.098,Z 228.149,A -85,B 0,C 180,E1 -25169.297,E2 -25169.297} C_VEL
LIN {X 0,Y 150.88,Z 223.731,A -85,B 0,C 180,E1 -25171.86,E2 -25171.86} C_VEL
LIN {X 0,Y 147.979,Z 219.672,A -85,B 0,C 180,E1 -25174.487,E2 -25174.487} C_VEL
LIN {X 0,Y 145.186,Z 216.481,A -85,B 0,C 180,E1 -25177.307,E2 -25177.307} C_VEL
LIN {X 0,Y 144.182,Z 214.773,A -85,B 0,C 180,E1 -25178.51,E2 -25178.51} C_VEL
LIN {X 0,Y 141.482,Z 212.128,A -85,B 0,C 180,E1 -25181.913,E2 -25181.913} C_VEL
LIN {X 0,Y 140.022,Z 209.401,A -85,B 0,C 180,E1 -25184.348,E2 -25184.348} C_VEL
LIN {X 0,Y 137.013,Z 206.96,A -85,B 0,C 180,E1 -25190.516,E2 -25190.516} C_VEL
LIN {X 0,Y 135.686,Z 204.091,A -85,B 0,C 180,E1 -25197.031,E2 -25197.031} C_VEL
LIN {X 0,Y 135.58,Z 203.616,A -85,B 0,C 180,E1 -25200.742,E2 -25200.742} C_VEL
LIN {X 0,Y 135.855,Z 204.669,A -85,B 0,C 180,E1 -25204.45,E2 -25204.45} C_VEL
LIN {X 0,Y 139.01,Z 208.907,A -85,B 0,C 180,E1 -25213.895,E2 -25213.895} C_VEL
LIN {X 0,Y 140.221,Z 209.681,A -85,B 0,C 180,E1 -25215.908,E2 -25215.908} C_VEL
LIN {X 0,Y 142.137,Z 213.02,A -85,B 0,C 180,E1 -25218.934,E2 -25218.934} C_VEL
LIN {X 0,Y 144.471,Z 215.174,A -85,B 0,C 180,E1 -25221.749,E2 -25221.749} C_VEL
LIN {X 0,Y 146.857,Z 218.671,A -85,B 0,C 180,E1 -25224.378,E2 -25224.378} C_VEL
